LIN {X 0,Y 185.523,Z 180.554,A -85,B 0,C 180,E1 -22370.264,E2 -22370.264} C_VEL
LIN {X 0,Y 186.732,Z 185.626,A -85,B 0,C 180,E1 -22372.872,E2 -22372.872} C_VEL
LIN {X 0,Y 194.907,Z 207.144,A -85,B 0,C 180,E1 -22375.125,E2 -22375.125} C_VEL
LIN {X 0,Y 199.126,Z 220.308,A -85,B 0,C 180,E1 -22376.315,E2 -22376.315} C_VEL
LIN {X 0,Y 201.437,Z 240.888,A -85,B 0,C 180,E1 -22377.565,E2 -22377.565} C_VEL
LIN {X 0,Y 199.217,Z 285.056,A -85,B 0,C 180,E1 -22379.362,E2 -22379.362} C_VEL
LIN {X 0,Y 198.176,Z 290.854,A -85,B 0,C 180,E1 -22379.532,E2 -22379.532} C_VEL
LIN {X 0,Y 194.625,Z 300.116,A -85,B 0,C 180,E1 -22379.764,E2 -22379.764} C_VEL
LIN {X 0,Y 190.969,Z 309.221,A -85,B 0,C 180,E1 -22380.201,E2 -22380.201} C_VEL
LIN {X 0,Y 189.736,Z 314.767,A -85,B 0,C 180,E1 -22380.703,E2 -22380.703} C_VEL
LIN {X 0,Y 187.977,Z 326.317,A -85,B 0,C 180,E1 -22382.138,E2 -22382.138} C_VEL
LIN {X 0,Y 185.921,Z 337.434,A -85,B 0,C 180,E1 -22383.932,E2 -22383.932} C_VEL
LIN {X 0,Y 183.615,Z 348.891,A -85,B 0,C 180,E1 -22386.303,E2 -22386.303} C_VEL
LIN {X 0,Y 181.324,Z 359.447,A -85,B 0,C 180,E1 -22389.126,E2 -22389.126} C_VEL
LIN {X 0,Y 179.446,Z 368.889,A -85,B 0,C 180,E1 -22392.33,E2 -22392.33} C_VEL
LIN {X 0,Y 177.807,Z 376.667,A -85,B 0,C 180,E1 -22395.698,E2 -22395.698} C_VEL
LIN {X 0,Y 176.949,Z 381.981,A -85,B 0,C 180,E1 -22398.545,E2 -22398.545} C_VEL
LIN {X 0,Y 176.345,Z 387.087,A -85,B 0,C 180,E1 -22401.982,E2 -22401.982} C_VEL
LIN {X 0,Y 176.061,Z 390.987,A -85,B 0,C 180,E1 -22405.421,E2 -22405.421} C_VEL
LIN {X 0,Y 176.043,Z 392.971,A -85,B 0,C 180,E1 -22407.712,E2 -22407.712} C_VEL
LIN {X 0,Y 176.191,Z 394.524,A -85,B 0,C 180,E1 -22410,E2 -22410} C_VEL
LIN {X 0,Y 175.998,Z 395.943,A -85,B 0,C 180,E1 -22413.319,E2 -22413.319} C_VEL
LIN {X 0,Y 176.144,Z 396.529,A -85,B 0,C 180,E1 -22416.874,E2 -22416.874} C_VEL
LIN {X 0,Y 177.087,Z 395.919,A -85,B 0,C 180,E1 -22421.445,E2 -22421.445} C_VEL
LIN {X 0,Y 178.986,Z 393.704,A -85,B 0,C 180,E1 -22425.953,E2 -22425.953} C_VEL
LIN {X 0,Y 181.258,Z 391.001,A -85,B 0,C 180,E1 -22429.242,E2 -22429.242} C_VEL
LIN {X 0,Y 184.177,Z 387.313,A -85,B 0,C 180,E1 -22432.431,E2 -22432.431} C_VEL
LIN {X 0,Y 187.917,Z 381.869,A -85,B 0,C 180,E1 -22435.953,E2 -22435.953} C_VEL
LIN {X 0,Y 192.068,Z 375.591,A -85,B 0,C 180,E1 -22439.001,E2 -22439.001} C_VEL
LIN {X 0,Y 196.577,Z 368.083,A -85,B 0,C 180,E1 -22441.825,E2 -22441.825} C_VEL
LIN {X 0,Y 201.898,Z 358.701,A -85,B 0,C 180,E1 -22444.447,E2 -22444.447} C_VEL
LIN {X 0,Y 207.006,Z 348.132,A -85,B 0,C 180,E1 -22446.753,E2 -22446.753} C_VEL
LIN {X 0,Y 211.458,Z 337.471,A -85,B 0,C 180,E1 -22448.547,E2 -22448.547} C_VEL
LIN {X 0,Y 215.19,Z 327.2,A -85,B 0,C 180,E1 -22449.861,E2 -22449.861} C_VEL
LIN {X 0,Y 219.022,Z 314.154,A -85,B 0,C 180,E1 -22451.132,E2 -22451.132} C_VEL
LIN {X 0,Y 221.965,Z 300.978,A -85,B 0,C 180,E1 -22452.032,E2 -22452.032} C_VEL
LIN {X 0,Y 224.04,Z 287.051,A -85,B 0,C 180,E1 -22452.66,E2 -22452.66} C_VEL
LIN {X 0,Y 227.25,Z 253.842,A -85,B 0,C 180,E1 -22453.843,E2 -22453.843} C_VEL
LIN {X 0,Y 223.841,Z 244.653,A -85,B 0,C 180,E1 -22456.051,E2 -22456.051} C_VEL
LIN {X 0,Y 220.21,Z 236.597,A -85,B 0,C 180,E1 -22458.58,E2 -22458.58} C_VEL
LIN {X 0,Y 217.139,Z 230.6,A -85,B 0,C 180,E1 -22461.012,E2 -22461.012} C_VEL
LIN {X 0,Y 214.883,Z 226.367,A -85,B 0,C 180,E1 -22463.117,E2 -22463.117} C_VEL
LIN {X 0,Y 212.143,Z 221.304,A -85,B 0,C 180,E1 -22466.228,E2 -22466.228} C_VEL
LIN {X 0,Y 208.997,Z 215.881,A -85,B 0,C 180,E1 -22471.764,E2 -22471.764} C_VEL
LIN {X 0,Y 208.244,Z 214.671,A -85,B 0,C 180,E1 -22474.351,E2 -22474.351} C_VEL
LIN {X 0,Y 207.997,Z 214.147,A -85,B 0,C 180,E1 -22478.18,E2 -22478.18} C_VEL
LIN {X 0,Y 208.898,Z 214.551,A -85,B 0,C 180,E1 -22482.075,E2 -22482.075} C_VEL
LIN {X 0,Y 212.652,Z 219.409,A -85,B 0,C 180,E1 -22488.471,E2 -22488.471} C_VEL
LIN {X 0,Y 215.724,Z 224.28,A -85,B 0,C 180,E1 -22491.751,E2 -22491.751} C_VEL
LIN {X 0,Y 218.763,Z 228.903,A -85,B 0,C 180,E1 -22494.313,E2 -22494.313} C_VEL
LIN {X 0,Y 221.395,Z 233.953,A -85,B 0,C 180,E1 -22496.315,E2 -22496.315} C_VEL
LIN {X 0,Y 225.254,Z 241.753,A -85,B 0,C 180,E1 -22498.857,E2 -22498.857} C_VEL
LIN {X 0,Y 227.673,Z 247.671,A -85,B 0,C 180,E1 -22500.375,E2 -22500.375} C_VEL
LIN {X 0,Y 223.79,Z 286.154,A -85,B 0,C 180,E1 -22501.764,E2 -22501.764} C_VEL
LIN {X 0,Y 221.454,Z 299.905,A -85,B 0,C 180,E1 -22502.557,E2 -22502.557} C_VEL
LIN {X 0,Y 218.622,Z 311.882,A -85,B 0,C 180,E1 -22503.551,E2 -22503.551} C_VEL
LIN {X 0,Y 214.983,Z 323.909,A -85,B 0,C 180,E1 -22504.922,E2 -22504.922} C_VEL
LIN {X 0,Y 210.876,Z 334.991,A -85,B 0,C 180,E1 -22506.567,E2 -22506.567} C_VEL
LIN {X 0,Y 206.146,Z 345.721,A -85,B 0,C 180,E1 -22508.638,E2 -22508.638} C_VEL
LIN {X 0,Y 201.058,Z 355.6,A -85,B 0,C 180,E1 -22511.104,E2 -22511.104} C_VEL
LIN {X 0,Y 196.477,Z 363.559,A -85,B 0,C 180,E1 -22513.686,E2 -22513.686} C_VEL
LIN {X 0,Y 192.193,Z 370.197,A -85,B 0,C 180,E1 -22516.462,E2 -22516.462} C_VEL
LIN {X 0,Y 187.993,Z 376.022,A -85,B 0,C 180,E1 -22519.66,E2 -22519.66} C_VEL
LIN {X 0,Y 183.991,Z 381.142,A -85,B 0,C 180,E1 -22523.548,E2 -22523.548} C_VEL
LIN {X 0,Y 180.556,Z 384.879,A -85,B 0,C 180,E1 -22527.844,E2 -22527.844} C_VEL
LIN {X 0,Y 178.835,Z 386.437,A -85,B 0,C 180,E1 -22530.722,E2 -22530.722} C_VEL
LIN {X 0,Y 177.473,Z 387.301,A -85,B 0,C 180,E1 -22533.737,E2 -22533.737} C_VEL
LIN {X 0,Y 176.381,Z 387.452,A -85,B 0,C 180,E1 -22537.165,E2 -22537.165} C_VEL
LIN {X 0,Y 175.726,Z 386.737,A -85,B 0,C 180,E1 -22540.547,E2 -22540.547} C_VEL
LIN {X 0,Y 175.548,Z 385.172,A -85,B 0,C 180,E1 -22543.895,E2 -22543.895} C_VEL
LIN {X 0,Y 175.859,Z 381.648,A -85,B 0,C 180,E1 -22548.349,E2 -22548.349} C_VEL
LIN {X 0,Y 176.378,Z 377.958,A -85,B 0,C 180,E1 -22551.618,E2 -22551.618} C_VEL
LIN {X 0,Y 177.417,Z 371.966,A -85,B 0,C 180,E1 -22555.628,E2 -22555.628} C_VEL
LIN {X 0,Y 178.782,Z 364.796,A -85,B 0,C 180,E1 -22559.268,E2 -22559.268} C_VEL
LIN {X 0,Y 180.648,Z 355.985,A -85,B 0,C 180,E1 -22562.768,E2 -22562.768} C_VEL
LIN {X 0,Y 182.436,Z 347.714,A -85,B 0,C 180,E1 -22565.39,E2 -22565.39} C_VEL
LIN {X 0,Y 184.503,Z 337.858,A -85,B 0,C 180,E1 -22567.905,E2 -22567.905} C_VEL
LIN {X 0,Y 186.713,Z 326.401,A -85,B 0,C 180,E1 -22570.22,E2 -22570.22} C_VEL
LIN {X 0,Y 188.707,Z 314.366,A -85,B 0,C 180,E1 -22572.107,E2 -22572.107} C_VEL
LIN {X 0,Y 190.466,Z 301.472,A -85,B 0,C 180,E1 -22573.609,E2 -22573.609} C_VEL
LIN {X 0,Y 191.829,Z 288.229,A -85,B 0,C 180,E1 -22574.704,E2 -22574.704} C_VEL
LIN {X 0,Y 192.829,Z 272.096,A -85,B 0,C 180,E1 -22575.515,E2 -22575.515} C_VEL
LIN {X 0,Y 195.507,Z 223.333,A -85,B 0,C 180,E1 -22577.545,E2 -22577.545} C_VEL
LIN {X 0,Y 188.439,Z 202.79,A -85,B 0,C 180,E1 -22579.515,E2 -22579.515} C_VEL
LIN {X 0,Y 179.852,Z 183.966,A -85,B 0,C 180,E1 -22581.822,E2 -22581.822} C_VEL
LIN {X 0,Y 178.904,Z 181.199,A -85,B 0,C 180,E1 -22582.169,E2 -22582.169} C_VEL
LIN {X 0,Y 179.121,Z 181.175,A -85,B 0,C 180,E1 -22587.752,E2 -22587.752} C_VEL
LIN {X 0,Y 179.341,Z 181.15,A -85,B 0,C 180,E1 -22590,E2 -22590} C_VEL
LIN {X 0,Y 178.827,Z 181.214,A -85,B 0,C 180,E1 -22594.508,E2 -22594.508} C_VEL
LIN {X 0,Y 178.903,Z 181.203,A -85,B 0,C 180,E1 -22599.041,E2 -22599.041} C_VEL
LIN {X 0,Y 178.623,Z 181.236,A -85,B 0,C 180,E1 -22603.655,E2 -22603.655} C_VEL
LIN {X 0,Y 178.552,Z 181.244,A -85,B 0,C 180,E1 -22609.152,E2 -22609.152} C_VEL
LIN {X 0,Y 178.462,Z 181.253,A -85,B 0,C 180,E1 -22615.076,E2 -22615.076} C_VEL
LIN {X 0,Y 178.457,Z 181.247,A -85,B 0,C 180,E1 -22620.795,E2 -22620.795} C_VEL
LIN {X 0,Y 178.48,Z 181.247,A -85,B 0,C 180,E1 -22624.218,E2 -22624.218} C_VEL
LIN {X 0,Y 178.384,Z 181.263,A -85,B 0,C 180,E1 -22629.077,E2 -22629.077} C_VEL
LIN {X 0,Y 178.39,Z 181.25,A -85,B 0,C 180,E1 -22632.047,E2 -22632.047} C_VEL
LIN {X 0,Y 178.388,Z 181.253,A -85,B 0,C 180,E1 -22635.166,E2 -22635.166} C_VEL
LIN {X 0,Y 178.394,Z 181.261,A -85,B 0,C 180,E1 -22638.462,E2 -22638.462} C_VEL
LIN {X 0,Y 178.416,Z 181.251,A -85,B 0,C 180,E1 -22643.783,E2 -22643.783} C_VEL
LIN {X 0,Y 178.481,Z 181.231,A -85,B 0,C 180,E1 -22646.547,E2 -22646.547} C_VEL
LIN {X 0,Y 178.436,Z 181.255,A -85,B 0,C 180,E1 -22651.795,E2 -22651.795} C_VEL
LIN {X 0,Y 178.456,Z 181.251,A -85,B 0,C 180,E1 -22656.809,E2 -22656.809} C_VEL
LIN {X 0,Y 178.603,Z 181.212,A -85,B 0,C 180,E1 -22661.652,E2 -22661.652} C_VEL
LIN {X 0,Y 178.622,Z 181.23,A -85,B 0,C 180,E1 -22666.346,E2 -22666.346} C_VEL
LIN {X 0,Y 178.899,Z 181.193,A -85,B 0,C 180,E1 -22670.96,E2 -22670.96} C_VEL
LIN {X 0,Y 179.117,Z 181.163,A -85,B 0,C 180,E1 -22677.752,E2 -22677.752} C_VEL
LIN {X 0,Y 179.342,Z 181.143,A -85,B 0,C 180,E1 -22680.001,E2 -22680.001} C_VEL
LIN {X 0,Y 178.823,Z 181.202,A -85,B 0,C 180,E1 -22684.509,E2 -22684.509} C_VEL
LIN {X 0,Y 178.9,Z 181.193,A -85,B 0,C 180,E1 -22689.042,E2 -22689.042} C_VEL
LIN {X 0,Y 178.623,Z 181.234,A -85,B 0,C 180,E1 -22693.656,E2 -22693.656} C_VEL
LIN {X 0,Y 178.554,Z 181.241,A -85,B 0,C 180,E1 -22699.153,E2 -22699.153} C_VEL
LIN {X 0,Y 178.464,Z 181.249,A -85,B 0,C 180,E1 -22705.076,E2 -22705.076} C_VEL
LIN {X 0,Y 178.45,Z 181.252,A -85,B 0,C 180,E1 -22710.797,E2 -22710.797} C_VEL
LIN {X 0,Y 178.483,Z 181.236,A -85,B 0,C 180,E1 -22714.219,E2 -22714.219} C_VEL
LIN {X 0,Y 178.388,Z 181.264,A -85,B 0,C 180,E1 -22719.078,E2 -22719.078} C_VEL
LIN {X 0,Y 178.394,Z 181.264,A -85,B 0,C 180,E1 -22722.048,E2 -22722.048} C_VEL
LIN {X 0,Y 178.392,Z 181.264,A -85,B 0,C 180,E1 -22725.166,E2 -22725.166} C_VEL
LIN {X 0,Y 178.428,Z 181.35,A -85,B 0,C 180,E1 -22729.527,E2 -22729.527} C_VEL
LIN {X 0,Y 179.396,Z 185.381,A -85,B 0,C 180,E1 -22731.698,E2 -22731.698} C_VEL
LIN {X 0,Y 187.05,Z 205.093,A -85,B 0,C 180,E1 -22733.929,E2 -22733.929} C_VEL
LIN {X 0,Y 192.645,Z 221.29,A -85,B 0,C 180,E1 -22735.514,E2 -22735.514} C_VEL
LIN {X 0,Y 194.853,Z 241.898,A -85,B 0,C 180,E1 -22736.806,E2 -22736.806} C_VEL
LIN {X 0,Y 191.966,Z 293.825,A -85,B 0,C 180,E1 -22739.019,E2 -22739.019} C_VEL
LIN {X 0,Y 190.668,Z 307.543,A -85,B 0,C 180,E1 -22740.006,E2 -22740.006} C_VEL
LIN {X 0,Y 189.736,Z 314.767,A -85,B 0,C 180,E1 -22740.703,E2 -22740.703} C_VEL
LIN {X 0,Y 188.42,Z 320.204,A -85,B 0,C 180,E1 -22741.268,E2 -22741.268} C_VEL
LIN {X 0,Y 184.29,Z 328.708,A -85,B 0,C 180,E1 -22742.179,E2 -22742.179} C_VEL
LIN {X 0,Y 179.879,Z 336.864,A -85,B 0,C 180,E1 -22743.32,E2 -22743.32} C_VEL
LIN {X 0,Y 178.153,Z 341.765,A -85,B 0,C 180,E1 -22744.235,E2 -22744.235} C_VEL
LIN {X 0,Y 175.795,Z 352.848,A -85,B 0,C 180,E1 -22746.856,E2 -22746.856} C_VEL
LIN {X 0,Y 174.039,Z 361.107,A -85,B 0,C 180,E1 -22749.308,E2 -22749.308} C_VEL
LIN {X 0,Y 172.038,Z 370.429,A -85,B 0,C 180,E1 -22752.772,E2 -22752.772} C_VEL
LIN {X 0,Y 170.499,Z 377.896,A -85,B 0,C 180,E1 -22756.289,E2 -22756.289} C_VEL
LIN {X 0,Y 169.695,Z 382.937,A -85,B 0,C 180,E1 -22759.259,E2 -22759.259} C_VEL
LIN {X 0,Y 169.191,Z 387.794,A -85,B 0,C 180,E1 -22762.841,E2 -22762.841} C_VEL
LIN {X 0,Y 168.933,Z 391.821,A -85,B 0,C 180,E1 -22766.834,E2 -22766.834} C_VEL
LIN {X 0,Y 169.114,Z 394.051,A -85,B 0,C 180,E1 -22770,E2 -22770} C_VEL
LIN {X 0,Y 168.932,Z 395.495,A -85,B 0,C 180,E1 -22773.163,E2 -22773.163} C_VEL
LIN {X 0,Y 169.097,Z 396.296,A -85,B 0,C 180,E1 -22777.162,E2 -22777.162} C_VEL
LIN {X 0,Y 170.111,Z 395.823,A -85,B 0,C 180,E1 -22781.921,E2 -22781.921} C_VEL
LIN {X 0,Y 171.013,Z 395.023,A -85,B 0,C 180,E1 -22784.274,E2 -22784.274} C_VEL
LIN {X 0,Y 172.144,Z 393.803,A -85,B 0,C 180,E1 -22786.605,E2 -22786.605} C_VEL
LIN {X 0,Y 175.512,Z 390.163,A -85,B 0,C 180,E1 -22791.123,E2 -22791.123} C_VEL
LIN {X 0,Y 178.852,Z 386.299,A -85,B 0,C 180,E1 -22794.367,E2 -22794.367} C_VEL
LIN {X 0,Y 182.323,Z 381.399,A -85,B 0,C 180,E1 -22797.552,E2 -22797.552} C_VEL
LIN {X 0,Y 186.734,Z 375.257,A -85,B 0,C 180,E1 -22800.536,E2 -22800.536} C_VEL
LIN {X 0,Y 191.548,Z 367.741,A -85,B 0,C 180,E1 -22803.391,E2 -22803.391} C_VEL
LIN {X 0,Y 197.127,Z 358.396,A -85,B 0,C 180,E1 -22806.033,E2 -22806.033} C_VEL
LIN {X 0,Y 202.496,Z 347.857,A -85,B 0,C 180,E1 -22808.343,E2 -22808.343} C_VEL
LIN {X 0,Y 207.165,Z 337.161,A -85,B 0,C 180,E1 -22810.132,E2 -22810.132} C_VEL
LIN {X 0,Y 211.624,Z 325.18,A -85,B 0,C 180,E1 -22811.62,E2 -22811.62} C_VEL
LIN {X 0,Y 215.359,Z 312.674,A -85,B 0,C 180,E1 -22812.779,E2 -22812.779} C_VEL
LIN {X 0,Y 218.437,Z 298.841,A -85,B 0,C 180,E1 -22813.679,E2 -22813.679} C_VEL
LIN {X 0,Y 220.466,Z 284.829,A -85,B 0,C 180,E1 -22814.28,E2 -22814.28} C_VEL
LIN {X 0,Y 223.268,Z 256.597,A -85,B 0,C 180,E1 -22815.324,E2 -22815.324} C_VEL
LIN {X 0,Y 220.341,Z 248.569,A -85,B 0,C 180,E1 -22817.388,E2 -22817.388} C_VEL
LIN {X 0,Y 216.972,Z 240.885,A -85,B 0,C 180,E1 -22820.019,E2 -22820.019} C_VEL
LIN {X 0,Y 214.617,Z 236.021,A -85,B 0,C 180,E1 -22822.098,E2 -22822.098} C_VEL
LIN {X 0,Y 212.784,Z 232.436,A -85,B 0,C 180,E1 -22823.967,E2 -22823.967} C_VEL
LIN {X 0,Y 210.54,Z 227.94,A -85,B 0,C 180,E1 -22826.763,E2 -22826.763} C_VEL
LIN {X 0,Y 207.662,Z 222.626,A -85,B 0,C 180,E1 -22832.277,E2 -22832.277} C_VEL
LIN {X 0,Y 207.005,Z 221.519,A -85,B 0,C 180,E1 -22835.002,E2 -22835.002} C_VEL
LIN {X 0,Y 207.196,Z 221.214,A -85,B 0,C 180,E1 -22840.171,E2 -22840.171} C_VEL
LIN {X 0,Y 207.826,Z 221.735,A -85,B 0,C 180,E1 -22842.28,E2 -22842.28} C_VEL
LIN {X 0,Y 211.159,Z 226.339,A -85,B 0,C 180,E1 -22848.115,E2 -22848.115} C_VEL
LIN {X 0,Y 213.886,Z 230.84,A -85,B 0,C 180,E1 -22851.197,E2 -22851.197} C_VEL
LIN {X 0,Y 216.591,Z 235.183,A -85,B 0,C 180,E1 -22853.648,E2 -22853.648} C_VEL
LIN {X 0,Y 219.433,Z 241.032,A -85,B 0,C 180,E1 -22855.921,E2 -22855.921} C_VEL
LIN {X 0,Y 222.35,Z 247.28,A -85,B 0,C 180,E1 -22857.978,E2 -22857.978} C_VEL
LIN {X 0,Y 223.761,Z 251.117,A -85,B 0,C 180,E1 -22858.95,E2 -22858.95} C_VEL
LIN {X 0,Y 219.931,Z 286.55,A -85,B 0,C 180,E1 -22860.23,E2 -22860.23} C_VEL
LIN {X 0,Y 217.492,Z 300.162,A -85,B 0,C 180,E1 -22861.017,E2 -22861.017} C_VEL
LIN {X 0,Y 214.313,Z 312.803,A -85,B 0,C 180,E1 -22862.079,E2 -22862.079} C_VEL
LIN {X 0,Y 210.618,Z 324.429,A -85,B 0,C 180,E1 -22863.414,E2 -22863.414} C_VEL
LIN {X 0,Y 206.079,Z 336.077,A -85,B 0,C 180,E1 -22865.159,E2 -22865.159} C_VEL
LIN {X 0,Y 201.067,Z 346.77,A -85,B 0,C 180,E1 -22867.278,E2 -22867.278} C_VEL
LIN {X 0,Y 195.624,Z 356.675,A -85,B 0,C 180,E1 -22869.824,E2 -22869.824} C_VEL
LIN {X 0,Y 191.053,Z 364.048,A -85,B 0,C 180,E1 -22872.304,E2 -22872.304} C_VEL
LIN {X 0,Y 186.224,Z 371,A -85,B 0,C 180,E1 -22875.317,E2 -22875.317} C_VEL
LIN {X 0,Y 181.178,Z 377.479,A -85,B 0,C 180,E1 -22879.104,E2 -22879.104} C_VEL
LIN {X 0,Y 178.066,Z 381.099,A -85,B 0,C 180,E1 -22882.02,E2 -22882.02} C_VEL
LIN {X 0,Y 174.376,Z 384.854,A -85,B 0,C 180,E1 -22886.316,E2 -22886.316} C_VEL
LIN {X 0,Y 171.67,Z 386.998,A -85,B 0,C 180,E1 -22890.717,E2 -22890.717} C_VEL
LIN {X 0,Y 169.726,Z 387.734,A -85,B 0,C 180,E1 -22895.429,E2 -22895.429} C_VEL
LIN {X 0,Y 168.922,Z 387.306,A -85,B 0,C 180,E1 -22898.613,E2 -22898.613} C_VEL
LIN {X 0,Y 168.516,Z 386.174,A -85,B 0,C 180,E1 -22901.856,E2 -22901.856} C_VEL
LIN {X 0,Y 168.447,Z 384.252,A -85,B 0,C 180,E1 -22905.175,E2 -22905.175} C_VEL
LIN {X 0,Y 168.787,Z 381.419,A -85,B 0,C 180,E1 -22908.545,E2 -22908.545} C_VEL
LIN {X 0,Y 169.35,Z 377.474,A -85,B 0,C 180,E1 -22912.043,E2 -22912.043} C_VEL
LIN {X 0,Y 170.284,Z 372.225,A -85,B 0,C 180,E1 -22915.631,E2 -22915.631} C_VEL
LIN {X 0,Y 171.64,Z 365.335,A -85,B 0,C 180,E1 -22919.3,E2 -22919.3} C_VEL
LIN {X 0,Y 173.547,Z 356.471,A -85,B 0,C 180,E1 -22922.986,E2 -22922.986} C_VEL
LIN {X 0,Y 175.713,Z 346.879,A -85,B 0,C 180,E1 -22926.112,E2 -22926.112} C_VEL
LIN {X 0,Y 178.027,Z 336.047,A -85,B 0,C 180,E1 -22928.886,E2 -22928.886} C_VEL
LIN {X 0,Y 180.053,Z 325.747,A -85,B 0,C 180,E1 -22930.979,E2 -22930.979} C_VEL
LIN {X 0,Y 182.068,Z 313.748,A -85,B 0,C 180,E1 -22932.881,E2 -22932.881} C_VEL
LIN {X 0,Y 183.766,Z 301.825,A -85,B 0,C 180,E1 -22934.303,E2 -22934.303} C_VEL
LIN {X 0,Y 185.124,Z 288.738,A -85,B 0,C 180,E1 -22935.434,E2 -22935.434} C_VEL
LIN {X 0,Y 186.186,Z 273.821,A -85,B 0,C 180,E1 -22936.216,E2 -22936.216} C_VEL
LIN {X 0,Y 188.893,Z 224.499,A -85,B 0,C 180,E1 -22938.349,E2 -22938.349} C_VEL
LIN {X 0,Y 182.114,Z 204.991,A -85,B 0,C 180,E1 -22940.338,E2 -22940.338} C_VEL
LIN {X 0,Y 174.085,Z 187.342,A -85,B 0,C 180,E1 -22942.607,E2 -22942.607} C_VEL
LIN {X 0,Y 171.926,Z 182.6,A -85,B 0,C 180,E1 -22943.251,E2 -22943.251} C_VEL
LIN {X 0,Y 171.837,Z 182.08,A -85,B 0,C 180,E1 -22943.395,E2 -22943.395} C_VEL
LIN {X 0,Y 172.306,Z 182.026,A -85,B 0,C 180,E1 -22950,E2 -22950} C_VEL
LIN {X 0,Y 171.777,Z 182.092,A -85,B 0,C 180,E1 -22954.694,E2 -22954.694} C_VEL
LIN {X 0,Y 171.841,Z 182.084,A -85,B 0,C 180,E1 -22959.416,E2 -22959.416} C_VEL
LIN {X 0,Y 171.539,Z 182.119,A -85,B 0,C 180,E1 -22964.231,E2 -22964.231} C_VEL
LIN {X 0,Y 171.475,Z 182.126,A -85,B 0,C 180,E1 -22969.499,E2 -22969.499} C_VEL
LIN {X 0,Y 171.4,Z 182.134,A -85,B 0,C 180,E1 -22975.57,E2 -22975.57} C_VEL
LIN {X 0,Y 171.414,Z 182.125,A -85,B 0,C 180,E1 -22980.573,E2 -22980.573} C_VEL
LIN {X 0,Y 171.389,Z 182.132,A -85,B 0,C 180,E1 -22985.035,E2 -22985.035} C_VEL
LIN {X 0,Y 171.34,Z 182.141,A -85,B 0,C 180,E1 -22988.801,E2 -22988.801} C_VEL
LIN {X 0,Y 171.315,Z 182.129,A -85,B 0,C 180,E1 -22994.219,E2 -22994.219} C_VEL
LIN {X 0,Y 171.326,Z 182.144,A -85,B 0,C 180,E1 -22998.98,E2 -22998.98} C_VEL
LIN {X 0,Y 171.357,Z 182.136,A -85,B 0,C 180,E1 -23002.034,E2 -23002.034} C_VEL
LIN {X 0,Y 171.395,Z 182.118,A -85,B 0,C 180,E1 -23005.094,E2 -23005.094} C_VEL
LIN {X 0,Y 171.405,Z 182.127,A -85,B 0,C 180,E1 -23010.527,E2 -23010.527} C_VEL
LIN {X 0,Y 171.399,Z 182.132,A -85,B 0,C 180,E1 -23015.794,E2 -23015.794} C_VEL
LIN {X 0,Y 171.505,Z 182.096,A -85,B 0,C 180,E1 -23020.864,E2 -23020.864} C_VEL
LIN {X 0,Y 171.538,Z 182.11,A -85,B 0,C 180,E1 -23025.771,E2 -23025.771} C_VEL
LIN {X 0,Y 171.838,Z 182.074,A -85,B 0,C 180,E1 -23030.585,E2 -23030.585} C_VEL
LIN {X 0,Y 171.771,Z 182.066,A -85,B 0,C 180,E1 -23035.307,E2 -23035.307} C_VEL
LIN {X 0,Y 172.306,Z 182.019,A -85,B 0,C 180,E1 -23040.001,E2 -23040.001} C_VEL
LIN {X 0,Y 171.773,Z 182.079,A -85,B 0,C 180,E1 -23044.695,E2 -23044.695} C_VEL
LIN {X 0,Y 171.839,Z 182.073,A -85,B 0,C 180,E1 -23049.417,E2 -23049.417} C_VEL
LIN {X 0,Y 171.538,Z 182.114,A -85,B 0,C 180,E1 -23054.231,E2 -23054.231} C_VEL
LIN {X 0,Y 171.478,Z 182.124,A -85,B 0,C 180,E1 -23059.499,E2 -23059.499} C_VEL
LIN {X 0,Y 171.401,Z 182.131,A -85,B 0,C 180,E1 -23065.569,E2 -23065.569} C_VEL
LIN {X 0,Y 171.406,Z 182.131,A -85,B 0,C 180,E1 -23070.567,E2 -23070.567} C_VEL
LIN {X 0,Y 171.393,Z 182.123,A -85,B 0,C 180,E1 -23075.036,E2 -23075.036} C_VEL
LIN {X 0,Y 171.344,Z 182.142,A -85,B 0,C 180,E1 -23078.802,E2 -23078.802} C_VEL
LIN {X 0,Y 171.319,Z 182.146,A -85,B 0,C 180,E1 -23084.219,E2 -23084.219} C_VEL
LIN {X 0,Y 171.389,Z 182.155,A -85,B 0,C 180,E1 -23088.772,E2 -23088.772} C_VEL
LIN {X 0,Y 172.07,Z 185.224,A -85,B 0,C 180,E1 -23090.448,E2 -23090.448} C_VEL
LIN {X 0,Y 179.137,Z 202.761,A -85,B 0,C 180,E1 -23092.605,E2 -23092.605} C_VEL
LIN {X 0,Y 185.907,Z 222.273,A -85,B 0,C 180,E1 -23094.653,E2 -23094.653} C_VEL
LIN {X 0,Y 187.097,Z 229.819,A -85,B 0,C 180,E1 -23095.205,E2 -23095.205} C_VEL
LIN {X 0,Y 188.269,Z 242.646,A -85,B 0,C 180,E1 -23096.01,E2 -23096.01} C_VEL
LIN {X 0,Y 185.356,Z 293.514,A -85,B 0,C 180,E1 -23098.259,E2 -23098.259} C_VEL
LIN {X 0,Y 184.001,Z 307.3,A -85,B 0,C 180,E1 -23099.279,E2 -23099.279} C_VEL
LIN {X 0,Y 182.368,Z 319.378,A -85,B 0,C 180,E1 -23100.571,E2 -23100.571} C_VEL
LIN {X 0,Y 180.071,Z 331.931,A -85,B 0,C 180,E1 -23102.389,E2 -23102.389} C_VEL
LIN {X 0,Y 178.153,Z 341.765,A -85,B 0,C 180,E1 -23104.235,E2 -23104.235} C_VEL
LIN {X 0,Y 176.447,Z 346.538,A -85,B 0,C 180,E1 -23105.227,E2 -23105.227} C_VEL
LIN {X 0,Y 172.025,Z 353.866,A -85,B 0,C 180,E1 -23106.88,E2 -23106.88} C_VEL
LIN {X 0,Y 167.702,Z 360.692,A -85,B 0,C 180,E1 -23108.817,E2 -23108.817} C_VEL
LIN {X 0,Y 166.185,Z 364.652,A -85,B 0,C 180,E1 -23110.227,E2 -23110.227} C_VEL
LIN {X 0,Y 164.605,Z 371.946,A -85,B 0,C 180,E1 -23113.25,E2 -23113.25} C_VEL
LIN {X 0,Y 163.209,Z 379.043,A -85,B 0,C 180,E1 -23116.934,E2 -23116.934} C_VEL
LIN {X 0,Y 162.287,Z 385.506,A -85,B 0,C 180,E1 -23121.282,E2 -23121.282} C_VEL
LIN {X 0,Y 161.932,Z 389.689,A -85,B 0,C 180,E1 -23125.02,E2 -23125.02} C_VEL
LIN {X 0,Y 161.888,Z 391.867,A -85,B 0,C 180,E1 -23127.511,E2 -23127.511} C_VEL
LIN {X 0,Y 162.038,Z 393.549,A -85,B 0,C 180,E1 -23130,E2 -23130} C_VEL
LIN {X 0,Y 161.853,Z 394.955,A -85,B 0,C 180,E1 -23132.894,E2 -23132.894} C_VEL
LIN {X 0,Y 162.029,Z 396.059,A -85,B 0,C 180,E1 -23137.476,E2 -23137.476} C_VEL
LIN {X 0,Y 163.157,Z 395.723,A -85,B 0,C 180,E1 -23142.437,E2 -23142.437} C_VEL
LIN {X 0,Y 165.329,Z 393.897,A -85,B 0,C 180,E1 -23147.311,E2 -23147.311} C_VEL
LIN {X 0,Y 166.987,Z 392.384,A -85,B 0,C 180,E1 -23149.675,E2 -23149.675} C_VEL
LIN {X 0,Y 170.015,Z 389.345,A -85,B 0,C 180,E1 -23153.122,E2 -23153.122} C_VEL
LIN {X 0,Y 173.561,Z 385.303,A -85,B 0,C 180,E1 -23156.45,E2 -23156.45} C_VEL
LIN {X 0,Y 177.571,Z 380.206,A -85,B 0,C 180,E1 -23159.651,E2 -23159.651} C_VEL
LIN {X 0,Y 182.405,Z 373.865,A -85,B 0,C 180,E1 -23162.643,E2 -23162.643} C_VEL
LIN {X 0,Y 186.684,Z 367.498,A -85,B 0,C 180,E1 -23165.036,E2 -23165.036} C_VEL
LIN {X 0,Y 192.518,Z 358.143,A -85,B 0,C 180,E1 -23167.695,E2 -23167.695} C_VEL
LIN {X 0,Y 198.144,Z 347.584,A -85,B 0,C 180,E1 -23170.006,E2 -23170.006} C_VEL
LIN {X 0,Y 203.021,Z 336.957,A -85,B 0,C 180,E1 -23171.787,E2 -23171.787} C_VEL
LIN {X 0,Y 207.685,Z 325.055,A -85,B 0,C 180,E1 -23173.254,E2 -23173.254} C_VEL
LIN {X 0,Y 211.273,Z 313.725,A -85,B 0,C 180,E1 -23174.311,E2 -23174.311} C_VEL
LIN {X 0,Y 214.47,Z 300.41,A -85,B 0,C 180,E1 -23175.212,E2 -23175.212} C_VEL
LIN {X 0,Y 216.736,Z 286.356,A -85,B 0,C 180,E1 -23175.83,E2 -23175.83} C_VEL
LIN {X 0,Y 219.482,Z 259.569,A -85,B 0,C 180,E1 -23176.84,E2 -23176.84} C_VEL
LIN {X 0,Y 217.301,Z 253.29,A -85,B 0,C 180,E1 -23178.567,E2 -23178.567} C_VEL
LIN {X 0,Y 214.252,Z 246.021,A -85,B 0,C 180,E1 -23181.161,E2 -23181.161} C_VEL
LIN {X 0,Y 212.348,Z 241.789,A -85,B 0,C 180,E1 -23183.065,E2 -23183.065} C_VEL
LIN {X 0,Y 210.913,Z 238.821,A -85,B 0,C 180,E1 -23184.633,E2 -23184.633} C_VEL
LIN {X 0,Y 208.866,Z 234.483,A -85,B 0,C 180,E1 -23187.426,E2 -23187.426} C_VEL
LIN {X 0,Y 206.346,Z 229.374,A -85,B 0,C 180,E1 -23192.788,E2 -23192.788} C_VEL
LIN {X 0,Y 205.772,Z 228.371,A -85,B 0,C 180,E1 -23195.804,E2 -23195.804} C_VEL
LIN {X 0,Y 206.31,Z 228.334,A -85,B 0,C 180,E1 -23201.172,E2 -23201.172} C_VEL
LIN {X 0,Y 207.122,Z 229.711,A -85,B 0,C 180,E1 -23203.465,E2 -23203.465} C_VEL
LIN {X 0,Y 209.625,Z 233.092,A -85,B 0,C 180,E1 -23207.67,E2 -23207.67} C_VEL
LIN {X 0,Y 211.969,Z 237.247,A -85,B 0,C 180,E1 -23210.534,E2 -23210.534} C_VEL
LIN {X 0,Y 214.38,Z 241.282,A -85,B 0,C 180,E1 -23212.875,E2 -23212.875} C_VEL
LIN {X 0,Y 216.998,Z 247.043,A -85,B 0,C 180,E1 -23215.137,E2 -23215.137} C_VEL
LIN {X 0,Y 219.461,Z 252.674,A -85,B 0,C 180,E1 -23217.05,E2 -23217.05} C_VEL
LIN {X 0,Y 220.015,Z 254.15,A -85,B 0,C 180,E1 -23217.453,E2 -23217.453} C_VEL
LIN {X 0,Y 216.234,Z 287.473,A -85,B 0,C 180,E1 -23218.661,E2 -23218.661} C_VEL
LIN {X 0,Y 213.812,Z 300.27,A -85,B 0,C 180,E1 -23219.387,E2 -23219.387} C_VEL
LIN {X 0,Y 210.833,Z 311.927,A -85,B 0,C 180,E1 -23220.347,E2 -23220.347} C_VEL
LIN {X 0,Y 206.839,Z 324.068,A -85,B 0,C 180,E1 -23221.714,E2 -23221.714} C_VEL
LIN {X 0,Y 202.098,Z 335.694,A -85,B 0,C 180,E1 -23223.436,E2 -23223.436} C_VEL
LIN {X 0,Y 196.691,Z 346.702,A -85,B 0,C 180,E1 -23225.59,E2 -23225.59} C_VEL
LIN {X 0,Y 191.11,Z 356.456,A -85,B 0,C 180,E1 -23228.087,E2 -23228.087} C_VEL
LIN {X 0,Y 185.661,Z 364.773,A -85,B 0,C 180,E1 -23230.909,E2 -23230.909} C_VEL
LIN {X 0,Y 180.257,Z 371.983,A -85,B 0,C 180,E1 -23234.168,E2 -23234.168} C_VEL
LIN {X 0,Y 175.248,Z 377.911,A -85,B 0,C 180,E1 -23237.799,E2 -23237.799} C_VEL
LIN {X 0,Y 171.012,Z 382.398,A -85,B 0,C 180,E1 -23241.706,E2 -23241.706} C_VEL
LIN {X 0,Y 168.399,Z 384.806,A -85,B 0,C 180,E1 -23244.666,E2 -23244.666} C_VEL
LIN {X 0,Y 166.203,Z 386.5,A -85,B 0,C 180,E1 -23247.718,E2 -23247.718} C_VEL
LIN {X 0,Y 164.262,Z 387.621,A -85,B 0,C 180,E1 -23251.164,E2 -23251.164} C_VEL
LIN {X 0,Y 162.762,Z 387.939,A -85,B 0,C 180,E1 -23254.876,E2 -23254.876} C_VEL
LIN {X 0,Y 161.831,Z 387.357,A -85,B 0,C 180,E1 -23258.585,E2 -23258.585} C_VEL
LIN {X 0,Y 161.393,Z 385.904,A -85,B 0,C 180,E1 -23262.246,E2 -23262.246} C_VEL
LIN {X 0,Y 161.376,Z 383.631,A -85,B 0,C 180,E1 -23265.83,E2 -23265.83} C_VEL
LIN {X 0,Y 161.93,Z 379.421,A -85,B 0,C 180,E1 -23270.405,E2 -23270.405} C_VEL
LIN {X 0,Y 162.7,Z 374.955,A -85,B 0,C 180,E1 -23273.957,E2 -23273.957} C_VEL
LIN {X 0,Y 163.753,Z 369.334,A -85,B 0,C 180,E1 -23277.488,E2 -23277.488} C_VEL
LIN {X 0,Y 165.079,Z 363.009,A -85,B 0,C 180,E1 -23280.687,E2 -23280.687} C_VEL
LIN {X 0,Y 167.006,Z 354.548,A -85,B 0,C 180,E1 -23284.113,E2 -23284.113} C_VEL
LIN {X 0,Y 169.338,Z 344.57,A -85,B 0,C 180,E1 -23287.315,E2 -23287.315} C_VEL
LIN {X 0,Y 171.496,Z 334.758,A -85,B 0,C 180,E1 -23289.813,E2 -23289.813} C_VEL
LIN {X 0,Y 173.641,Z 323.774,A -85,B 0,C 180,E1 -23292.025,E2 -23292.025} C_VEL
LIN {X 0,Y 175.778,Z 311.181,A -85,B 0,C 180,E1 -23293.983,E2 -23293.983} C_VEL
LIN {X 0,Y 177.56,Z 298.182,A -85,B 0,C 180,E1 -23295.458,E2 -23295.458} C_VEL
LIN {X 0,Y 178.89,Z 283.878,A -85,B 0,C 180,E1 -23296.57,E2 -23296.57} C_VEL
LIN {X 0,Y 181.111,Z 248.12,A -85,B 0,C 180,E1 -23298.201,E2 -23298.201} C_VEL
LIN {X 0,Y 182.317,Z 225.866,A -85,B 0,C 180,E1 -23299.203,E2 -23299.203} C_VEL
LIN {X 0,Y 176.159,Z 208.076,A -85,B 0,C 180,E1 -23301.107,E2 -23301.107} C_VEL
LIN {X 0,Y 168.534,Z 191.154,A -85,B 0,C 180,E1 -23303.355,E2 -23303.355} C_VEL
LIN {X 0,Y 164.905,Z 183.853,A -85,B 0,C 180,E1 -23304.459,E2 -23304.459} C_VEL
LIN {X 0,Y 164.757,Z 182.963,A -85,B 0,C 180,E1 -23304.646,E2 -23304.646} C_VEL
LIN {X 0,Y 165.27,Z 182.903,A -85,B 0,C 180,E1 -23310,E2 -23310} C_VEL
LIN {X 0,Y 164.817,Z 182.957,A -85,B 0,C 180,E1 -23317.35,E2 -23317.35} C_VEL
LIN {X 0,Y 164.699,Z 182.972,A -85,B 0,C 180,E1 -23321.058,E2 -23321.058} C_VEL
LIN {X 0,Y 164.425,Z 183.003,A -85,B 0,C 180,E1 -23327.41,E2 -23327.41} C_VEL
LIN {X 0,Y 164.416,Z 183.003,A -85,B 0,C 180,E1 -23329.997,E2 -23329.997} C_VEL
LIN {X 0,Y 164.336,Z 183.014,A -85,B 0,C 180,E1 -23336.094,E2 -23336.094} C_VEL
LIN {X 0,Y 164.35,Z 183,A -85,B 0,C 180,E1 -23341.215,E2 -23341.215} C_VEL
LIN {X 0,Y 164.277,Z 183.021,A -85,B 0,C 180,E1 -23346.794,E2 -23346.794} C_VEL
LIN {X 0,Y 164.283,Z 183.015,A -85,B 0,C 180,E1 -23349.918,E2 -23349.918} C_VEL
LIN {X 0,Y 164.277,Z 183.003,A -85,B 0,C 180,E1 -23353.342,E2 -23353.342} C_VEL
LIN {X 0,Y 164.257,Z 183.018,A -85,B 0,C 180,E1 -23356.798,E2 -23356.798} C_VEL
LIN {X 0,Y 164.286,Z 183.02,A -85,B 0,C 180,E1 -23360.356,E2 -23360.356} C_VEL
LIN {X 0,Y 164.323,Z 183.003,A -85,B 0,C 180,E1 -23364.352,E2 -23364.352} C_VEL
LIN {X 0,Y 164.364,Z 182.997,A -85,B 0,C 180,E1 -23369.13,E2 -23369.13} C_VEL
LIN {X 0,Y 164.354,Z 183.012,A -85,B 0,C 180,E1 -23374.685,E2 -23374.685} C_VEL
LIN {X 0,Y 164.414,Z 182.983,A -85,B 0,C 180,E1 -23380.119,E2 -23380.119} C_VEL
LIN {X 0,Y 164.468,Z 182.99,A -85,B 0,C 180,E1 -23385.145,E2 -23385.145} C_VEL
LIN {X 0,Y 164.76,Z 182.958,A -85,B 0,C 180,E1 -23390.177,E2 -23390.177} C_VEL
LIN {X 0,Y 164.813,Z 182.941,A -85,B 0,C 180,E1 -23392.651,E2 -23392.651} C_VEL
LIN {X 0,Y 165.271,Z 182.895,A -85,B 0,C 180,E1 -23400.001,E2 -23400.001} C_VEL
LIN {X 0,Y 164.813,Z 182.938,A -85,B 0,C 180,E1 -23407.351,E2 -23407.351} C_VEL
LIN {X 0,Y 164.7,Z 182.967,A -85,B 0,C 180,E1 -23411.057,E2 -23411.057} C_VEL
LIN {X 0,Y 164.423,Z 182.993,A -85,B 0,C 180,E1 -23417.411,E2 -23417.411} C_VEL
LIN {X 0,Y 164.419,Z 183.006,A -85,B 0,C 180,E1 -23419.997,E2 -23419.997} C_VEL
LIN {X 0,Y 164.336,Z 183.016,A -85,B 0,C 180,E1 -23426.093,E2 -23426.093} C_VEL
LIN {X 0,Y 164.344,Z 183.004,A -85,B 0,C 180,E1 -23431.21,E2 -23431.21} C_VEL
LIN {X 0,Y 164.28,Z 183.019,A -85,B 0,C 180,E1 -23436.794,E2 -23436.794} C_VEL
LIN {X 0,Y 164.286,Z 183.018,A -85,B 0,C 180,E1 -23439.919,E2 -23439.919} C_VEL
LIN {X 0,Y 164.281,Z 183.022,A -85,B 0,C 180,E1 -23443.343,E2 -23443.343} C_VEL
LIN {X 0,Y 164.308,Z 183.027,A -85,B 0,C 180,E1 -23447.993,E2 -23447.993} C_VEL
LIN {X 0,Y 164.767,Z 185.015,A -85,B 0,C 180,E1 -23449.094,E2 -23449.094} C_VEL
LIN {X 0,Y 172.369,Z 203.596,A -85,B 0,C 180,E1 -23451.55,E2 -23451.55} C_VEL
LIN {X 0,Y 179.426,Z 223.731,A -85,B 0,C 180,E1 -23453.786,E2 -23453.786} C_VEL
LIN {X 0,Y 180.247,Z 228.001,A -85,B 0,C 180,E1 -23454.138,E2 -23454.138} C_VEL
LIN {X 0,Y 181.797,Z 242.264,A -85,B 0,C 180,E1 -23455.116,E2 -23455.116} C_VEL
LIN {X 0,Y 178.767,Z 293.265,A -85,B 0,C 180,E1 -23457.445,E2 -23457.445} C_VEL
LIN {X 0,Y 177.352,Z 307.043,A -85,B 0,C 180,E1 -23458.494,E2 -23458.494} C_VEL
LIN {X 0,Y 175.499,Z 320.162,A -85,B 0,C 180,E1 -23459.962,E2 -23459.962} C_VEL
LIN {X 0,Y 173.142,Z 332.485,A -85,B 0,C 180,E1 -23461.844,E2 -23461.844} C_VEL
LIN {X 0,Y 170.849,Z 343.677,A -85,B 0,C 180,E1 -23464.083,E2 -23464.083} C_VEL
LIN {X 0,Y 168.494,Z 354.193,A -85,B 0,C 180,E1 -23466.787,E2 -23466.787} C_VEL
LIN {X 0,Y 166.559,Z 362.99,A -85,B 0,C 180,E1 -23469.628,E2 -23469.628} C_VEL
LIN {X 0,Y 166.185,Z 364.652,A -85,B 0,C 180,E1 -23470.227,E2 -23470.227} C_VEL
LIN {X 0,Y 164.717,Z 368.493,A -85,B 0,C 180,E1 -23471.719,E2 -23471.719} C_VEL
LIN {X 0,Y 160.651,Z 374.032,A -85,B 0,C 180,E1 -23474.219,E2 -23474.219} C_VEL
LIN {X 0,Y 156.758,Z 379.046,A -85,B 0,C 180,E1 -23476.986,E2 -23476.986} C_VEL
LIN {X 0,Y 155.601,Z 381.869,A -85,B 0,C 180,E1 -23478.852,E2 -23478.852} C_VEL
LIN {X 0,Y 154.973,Z 387.667,A -85,B 0,C 180,E1 -23483.49,E2 -23483.49} C_VEL
LIN {X 0,Y 154.818,Z 391.24,A -85,B 0,C 180,E1 -23487.398,E2 -23487.398} C_VEL
LIN {X 0,Y 154.945,Z 393.044,A -85,B 0,C 180,E1 -23490,E2 -23490} C_VEL
LIN {X 0,Y 154.795,Z 394.402,A -85,B 0,C 180,E1 -23492.733,E2 -23492.733} C_VEL
LIN {X 0,Y 154.975,Z 395.768,A -85,B 0,C 180,E1 -23497.819,E2 -23497.819} C_VEL
LIN {X 0,Y 155.45,Z 395.905,A -85,B 0,C 180,E1 -23500.418,E2 -23500.418} C_VEL
LIN {X 0,Y 157.229,Z 394.979,A -85,B 0,C 180,E1 -23505.556,E2 -23505.556} C_VEL
LIN {X 0,Y 158.545,Z 393.954,A -85,B 0,C 180,E1 -23508.076,E2 -23508.076} C_VEL
LIN {X 0,Y 160.304,Z 392.547,A -85,B 0,C 180,E1 -23510.531,E2 -23510.531} C_VEL
LIN {X 0,Y 163.526,Z 389.642,A -85,B 0,C 180,E1 -23514.097,E2 -23514.097} C_VEL
LIN {X 0,Y 167.228,Z 385.792,A -85,B 0,C 180,E1 -23517.534,E2 -23517.534} C_VEL
LIN {X 0,Y 171.487,Z 380.892,A -85,B 0,C 180,E1 -23520.815,E2 -23520.815} C_VEL
LIN {X 0,Y 177.357,Z 373.648,A -85,B 0,C 180,E1 -23524.379,E2 -23524.379} C_VEL
LIN {X 0,Y 181.98,Z 367.256,A -85,B 0,C 180,E1 -23526.769,E2 -23526.769} C_VEL
LIN {X 0,Y 188.084,Z 357.975,A -85,B 0,C 180,E1 -23529.436,E2 -23529.436} C_VEL
LIN {X 0,Y 193.986,Z 347.507,A -85,B 0,C 180,E1 -23531.736,E2 -23531.736} C_VEL
LIN {X 0,Y 199.073,Z 336.918,A -85,B 0,C 180,E1 -23533.504,E2 -23533.504} C_VEL
LIN {X 0,Y 203.922,Z 325.035,A -85,B 0,C 180,E1 -23534.951,E2 -23534.951} C_VEL
LIN {X 0,Y 207.656,Z 313.728,A -85,B 0,C 180,E1 -23535.987,E2 -23535.987} C_VEL
LIN {X 0,Y 210.956,Z 300.587,A -85,B 0,C 180,E1 -23536.869,E2 -23536.869} C_VEL
LIN {X 0,Y 213.38,Z 286.214,A -85,B 0,C 180,E1 -23537.507,E2 -23537.507} C_VEL
LIN {X 0,Y 215.96,Z 262.719,A -85,B 0,C 180,E1 -23538.387,E2 -23538.387} C_VEL
LIN {X 0,Y 213.546,Z 255.837,A -85,B 0,C 180,E1 -23540.528,E2 -23540.528} C_VEL
LIN {X 0,Y 210.959,Z 249.317,A -85,B 0,C 180,E1 -23543.153,E2 -23543.153} C_VEL
LIN {X 0,Y 209.068,Z 245.223,A -85,B 0,C 180,E1 -23545.328,E2 -23545.328} C_VEL
LIN {X 0,Y 207.263,Z 241.039,A -85,B 0,C 180,E1 -23548.045,E2 -23548.045} C_VEL
LIN {X 0,Y 205.062,Z 236.181,A -85,B 0,C 180,E1 -23553.248,E2 -23553.248} C_VEL
LIN {X 0,Y 204.552,Z 235.246,A -85,B 0,C 180,E1 -23556.935,E2 -23556.935} C_VEL
LIN {X 0,Y 205.262,Z 235.446,A -85,B 0,C 180,E1 -23561.491,E2 -23561.491} C_VEL
LIN {X 0,Y 208.083,Z 239.855,A -85,B 0,C 180,E1 -23567.199,E2 -23567.199} C_VEL
LIN {X 0,Y 210.174,Z 243.813,A -85,B 0,C 180,E1 -23569.962,E2 -23569.962} C_VEL
LIN {X 0,Y 212.402,Z 247.708,A -85,B 0,C 180,E1 -23572.241,E2 -23572.241} C_VEL
LIN {X 0,Y 215.867,Z 255.837,A -85,B 0,C 180,E1 -23575.374,E2 -23575.374} C_VEL
LIN {X 0,Y 216.503,Z 257.473,A -85,B 0,C 180,E1 -23575.901,E2 -23575.901} C_VEL
LIN {X 0,Y 212.847,Z 287.795,A -85,B 0,C 180,E1 -23577.001,E2 -23577.001} C_VEL
LIN {X 0,Y 210.138,Z 301.305,A -85,B 0,C 180,E1 -23577.769,E2 -23577.769} C_VEL
LIN {X 0,Y 206.436,Z 314.566,A -85,B 0,C 180,E1 -23578.902,E2 -23578.902} C_VEL
LIN {X 0,Y 202.376,Z 326.059,A -85,B 0,C 180,E1 -23580.248,E2 -23580.248} C_VEL
LIN {X 0,Y 197.25,Z 337.746,A -85,B 0,C 180,E1 -23582.041,E2 -23582.041} C_VEL
LIN {X 0,Y 191.641,Z 348.384,A -85,B 0,C 180,E1 -23584.205,E2 -23584.205} C_VEL
LIN {X 0,Y 186.298,Z 357.078,A -85,B 0,C 180,E1 -23586.497,E2 -23586.497} C_VEL
LIN {X 0,Y 181.307,Z 364.231,A -85,B 0,C 180,E1 -23588.919,E2 -23588.919} C_VEL
LIN {X 0,Y 175.871,Z 371.189,A -85,B 0,C 180,E1 -23591.974,E2 -23591.974} C_VEL
LIN {X 0,Y 170.678,Z 377.08,A -85,B 0,C 180,E1 -23595.47,E2 -23595.47} C_VEL
LIN {X 0,Y 165.376,Z 382.317,A -85,B 0,C 180,E1 -23599.874,E2 -23599.874} C_VEL
LIN {X 0,Y 161.578,Z 385.482,A -85,B 0,C 180,E1 -23604.021,E2 -23604.021} C_VEL
LIN {X 0,Y 158.906,Z 387.258,A -85,B 0,C 180,E1 -23607.807,E2 -23607.807} C_VEL
LIN {X 0,Y 156.46,Z 388.131,A -85,B 0,C 180,E1 -23612.616,E2 -23612.616} C_VEL
LIN {X 0,Y 155.274,Z 387.933,A -85,B 0,C 180,E1 -23616.042,E2 -23616.042} C_VEL
LIN {X 0,Y 154.57,Z 387,A -85,B 0,C 180,E1 -23619.534,E2 -23619.534} C_VEL
LIN {X 0,Y 154.253,Z 385.256,A -85,B 0,C 180,E1 -23623.2,E2 -23623.2} C_VEL
LIN {X 0,Y 154.384,Z 382.629,A -85,B 0,C 180,E1 -23626.935,E2 -23626.935} C_VEL
LIN {X 0,Y 155.04,Z 378.181,A -85,B 0,C 180,E1 -23631.444,E2 -23631.444} C_VEL
LIN {X 0,Y 156.103,Z 372.24,A -85,B 0,C 180,E1 -23635.893,E2 -23635.893} C_VEL
LIN {X 0,Y 157.65,Z 364.819,A -85,B 0,C 180,E1 -23640.102,E2 -23640.102} C_VEL
LIN {X 0,Y 159.596,Z 356.338,A -85,B 0,C 180,E1 -23643.874,E2 -23643.874} C_VEL
LIN {X 0,Y 162.048,Z 346.24,A -85,B 0,C 180,E1 -23647.363,E2 -23647.363} C_VEL
LIN {X 0,Y 164.536,Z 335.32,A -85,B 0,C 180,E1 -23650.325,E2 -23650.325} C_VEL
LIN {X 0,Y 166.65,Z 325.046,A -85,B 0,C 180,E1 -23652.514,E2 -23652.514} C_VEL
LIN {X 0,Y 168.883,Z 312.581,A -85,B 0,C 180,E1 -23654.568,E2 -23654.568} C_VEL
LIN {X 0,Y 170.668,Z 300.478,A -85,B 0,C 180,E1 -23656.063,E2 -23656.063} C_VEL
LIN {X 0,Y 172.088,Z 287.234,A -85,B 0,C 180,E1 -23657.206,E2 -23657.206} C_VEL
LIN {X 0,Y 173.254,Z 270.409,A -85,B 0,C 180,E1 -23658.098,E2 -23658.098} C_VEL
LIN {X 0,Y 175.931,Z 227.786,A -85,B 0,C 180,E1 -23660.054,E2 -23660.054} C_VEL
LIN {X 0,Y 170.393,Z 211.538,A -85,B 0,C 180,E1 -23661.843,E2 -23661.843} C_VEL
LIN {X 0,Y 162.232,Z 193.323,A -85,B 0,C 180,E1 -23664.395,E2 -23664.395} C_VEL
LIN {X 0,Y 157.883,Z 184.669,A -85,B 0,C 180,E1 -23665.812,E2 -23665.812} C_VEL
LIN {X 0,Y 157.746,Z 183.838,A -85,B 0,C 180,E1 -23666.009,E2 -23666.009} C_VEL
LIN {X 0,Y 158.233,Z 183.78,A -85,B 0,C 180,E1 -23670,E2 -23670} C_VEL
LIN {X 0,Y 157.755,Z 183.838,A -85,B 0,C 180,E1 -23677.681,E2 -23677.681} C_VEL
LIN {X 0,Y 157.628,Z 183.853,A -85,B 0,C 180,E1 -23681.224,E2 -23681.224} C_VEL
LIN {X 0,Y 157.403,Z 183.881,A -85,B 0,C 180,E1 -23685.539,E2 -23685.539} C_VEL
LIN {X 0,Y 157.299,Z 183.888,A -85,B 0,C 180,E1 -23690.943,E2 -23690.943} C_VEL
LIN {X 0,Y 157.263,Z 183.895,A -85,B 0,C 180,E1 -23696.65,E2 -23696.65} C_VEL
LIN {X 0,Y 157.261,Z 183.881,A -85,B 0,C 180,E1 -23702.431,E2 -23702.431} C_VEL
LIN {X 0,Y 157.255,Z 183.895,A -85,B 0,C 180,E1 -23706.445,E2 -23706.445} C_VEL
LIN {X 0,Y 157.186,Z 183.889,A -85,B 0,C 180,E1 -23712.119,E2 -23712.119} C_VEL
LIN {X 0,Y 157.186,Z 183.902,A -85,B 0,C 180,E1 -23717.883,E2 -23717.883} C_VEL
LIN {X 0,Y 157.256,Z 183.886,A -85,B 0,C 180,E1 -23723.557,E2 -23723.557} C_VEL
LIN {X 0,Y 157.277,Z 183.874,A -85,B 0,C 180,E1 -23728.105,E2 -23728.105} C_VEL
LIN {X 0,Y 157.264,Z 183.894,A -85,B 0,C 180,E1 -23733.457,E2 -23733.457} C_VEL
LIN {X 0,Y 157.357,Z 183.865,A -85,B 0,C 180,E1 -23739.704,E2 -23739.704} C_VEL
LIN {X 0,Y 157.402,Z 183.865,A -85,B 0,C 180,E1 -23744.462,E2 -23744.462} C_VEL
LIN {X 0,Y 157.683,Z 183.839,A -85,B 0,C 180,E1 -23749.731,E2 -23749.731} C_VEL
LIN {X 0,Y 157.752,Z 183.822,A -85,B 0,C 180,E1 -23752.32,E2 -23752.32} C_VEL
LIN {X 0,Y 158.233,Z 183.771,A -85,B 0,C 180,E1 -23760.001,E2 -23760.001} C_VEL
LIN {X 0,Y 157.753,Z 183.818,A -85,B 0,C 180,E1 -23767.682,E2 -23767.682} C_VEL
LIN {X 0,Y 157.629,Z 183.848,A -85,B 0,C 180,E1 -23771.223,E2 -23771.223} C_VEL
LIN {X 0,Y 157.401,Z 183.87,A -85,B 0,C 180,E1 -23775.541,E2 -23775.541} C_VEL
LIN {X 0,Y 157.302,Z 183.891,A -85,B 0,C 180,E1 -23780.943,E2 -23780.943} C_VEL
LIN {X 0,Y 157.267,Z 183.896,A -85,B 0,C 180,E1 -23786.65,E2 -23786.65} C_VEL
LIN {X 0,Y 157.261,Z 183.878,A -85,B 0,C 180,E1 -23792.432,E2 -23792.432} C_VEL
LIN {X 0,Y 157.259,Z 183.892,A -85,B 0,C 180,E1 -23796.445,E2 -23796.445} C_VEL
LIN {X 0,Y 157.19,Z 183.905,A -85,B 0,C 180,E1 -23802.119,E2 -23802.119} C_VEL
LIN {X 0,Y 157.229,Z 183.937,A -85,B 0,C 180,E1 -23807.188,E2 -23807.188} C_VEL
LIN {X 0,Y 157.444,Z 184.823,A -85,B 0,C 180,E1 -23807.622,E2 -23807.622} C_VEL
LIN {X 0,Y 165.494,Z 204.029,A -85,B 0,C 180,E1 -23810.383,E2 -23810.383} C_VEL
LIN {X 0,Y 171.492,Z 220.863,A -85,B 0,C 180,E1 -23812.392,E2 -23812.392} C_VEL
LIN {X 0,Y 173.752,Z 228.226,A -85,B 0,C 180,E1 -23813.161,E2 -23813.161} C_VEL
LIN {X 0,Y 175.245,Z 243.526,A -85,B 0,C 180,E1 -23814.231,E2 -23814.231} C_VEL
LIN {X 0,Y 172.116,Z 293.915,A -85,B 0,C 180,E1 -23816.635,E2 -23816.635} C_VEL
LIN {X 0,Y 170.656,Z 307.399,A -85,B 0,C 180,E1 -23817.718,E2 -23817.718} C_VEL
LIN {X 0,Y 168.834,Z 319.831,A -85,B 0,C 180,E1 -23819.168,E2 -23819.168} C_VEL
LIN {X 0,Y 166.267,Z 332.942,A -85,B 0,C 180,E1 -23821.261,E2 -23821.261} C_VEL
LIN {X 0,Y 163.887,Z 343.977,A -85,B 0,C 180,E1 -23823.582,E2 -23823.582} C_VEL
LIN {X 0,Y 161.388,Z 354.709,A -85,B 0,C 180,E1 -23826.5,E2 -23826.5} C_VEL
LIN {X 0,Y 159.119,Z 364.744,A -85,B 0,C 180,E1 -23829.983,E2 -23829.983} C_VEL
LIN {X 0,Y 157.181,Z 373.228,A -85,B 0,C 180,E1 -23833.772,E2 -23833.772} C_VEL
LIN {X 0,Y 155.884,Z 380.041,A -85,B 0,C 180,E1 -23837.634,E2 -23837.634} C_VEL
LIN {X 0,Y 155.601,Z 381.869,A -85,B 0,C 180,E1 -23838.852,E2 -23838.852} C_VEL
LIN {X 0,Y 154.561,Z 384.477,A -85,B 0,C 180,E1 -23840.782,E2 -23840.782} C_VEL
LIN {X 0,Y 151.313,Z 388.013,A -85,B 0,C 180,E1 -23844.044,E2 -23844.044} C_VEL
LIN {X 0,Y 148.814,Z 390.316,A -85,B 0,C 180,E1 -23846.813,E2 -23846.813} C_VEL
LIN {X 0,Y 147.87,Z 391.846,A -85,B 0,C 180,E1 -23849.005,E2 -23849.005} C_VEL
LIN {X 0,Y 147.849,Z 392.308,A -85,B 0,C 180,E1 -23849.748,E2 -23849.748} C_VEL
LIN {X 0,Y 147.718,Z 393.897,A -85,B 0,C 180,E1 -23852.727,E2 -23852.727} C_VEL
LIN {X 0,Y 147.944,Z 395.458,A -85,B 0,C 180,E1 -23858.193,E2 -23858.193} C_VEL
LIN {X 0,Y 149.262,Z 395.515,A -85,B 0,C 180,E1 -23863.616,E2 -23863.616} C_VEL
LIN {X 0,Y 151.798,Z 394.016,A -85,B 0,C 180,E1 -23868.91,E2 -23868.91} C_VEL
LIN {X 0,Y 155.863,Z 390.992,A -85,B 0,C 180,E1 -23873.941,E2 -23873.941} C_VEL
LIN {X 0,Y 159.712,Z 387.623,A -85,B 0,C 180,E1 -23877.518,E2 -23877.518} C_VEL
LIN {X 0,Y 163.839,Z 383.274,A -85,B 0,C 180,E1 -23880.98,E2 -23880.98} C_VEL
LIN {X 0,Y 168.913,Z 377.792,A -85,B 0,C 180,E1 -23884.172,E2 -23884.172} C_VEL
LIN {X 0,Y 174.367,Z 371.085,A -85,B 0,C 180,E1 -23887.198,E2 -23887.198} C_VEL
LIN {X 0,Y 180.621,Z 362.771,A -85,B 0,C 180,E1 -23889.941,E2 -23889.941} C_VEL
LIN {X 0,Y 187.192,Z 352.452,A -85,B 0,C 180,E1 -23892.515,E2 -23892.515} C_VEL
LIN {X 0,Y 192.914,Z 341.871,A -85,B 0,C 180,E1 -23894.529,E2 -23894.529} C_VEL
LIN {X 0,Y 197.849,Z 331.38,A -85,B 0,C 180,E1 -23895.997,E2 -23895.997} C_VEL
LIN {X 0,Y 202.273,Z 319.963,A -85,B 0,C 180,E1 -23897.22,E2 -23897.22} C_VEL
LIN {X 0,Y 206.198,Z 307.268,A -85,B 0,C 180,E1 -23898.208,E2 -23898.208} C_VEL
LIN {X 0,Y 209.144,Z 293.927,A -85,B 0,C 180,E1 -23898.931,E2 -23898.931} C_VEL
LIN {X 0,Y 211.858,Z 272.966,A -85,B 0,C 180,E1 -23899.726,E2 -23899.726} C_VEL
LIN {X 0,Y 212.616,Z 265.891,A -85,B 0,C 180,E1 -23900.018,E2 -23900.018} C_VEL
LIN {X 0,Y 210.203,Z 258.849,A -85,B 0,C 180,E1 -23902.484,E2 -23902.484} C_VEL
LIN {X 0,Y 208.319,Z 254.079,A -85,B 0,C 180,E1 -23904.659,E2 -23904.659} C_VEL
LIN {X 0,Y 207.115,Z 251.189,A -85,B 0,C 180,E1 -23906.306,E2 -23906.306} C_VEL
LIN {X 0,Y 205.673,Z 247.635,A -85,B 0,C 180,E1 -23908.677,E2 -23908.677} C_VEL
LIN {X 0,Y 203.89,Z 243.206,A -85,B 0,C 180,E1 -23913.377,E2 -23913.377} C_VEL
LIN {X 0,Y 203.432,Z 242.26,A -85,B 0,C 180,E1 -23916.8,E2 -23916.8} C_VEL
LIN {X 0,Y 204.091,Z 242.454,A -85,B 0,C 180,E1 -23921.381,E2 -23921.381} C_VEL
LIN {X 0,Y 206.55,Z 246.593,A -85,B 0,C 180,E1 -23926.711,E2 -23926.711} C_VEL
LIN {X 0,Y 208.298,Z 250.106,A -85,B 0,C 180,E1 -23929.222,E2 -23929.222} C_VEL
LIN {X 0,Y 210.5,Z 254.236,A -85,B 0,C 180,E1 -23931.647,E2 -23931.647} C_VEL
LIN {X 0,Y 213.119,Z 261.018,A -85,B 0,C 180,E1 -23934.277,E2 -23934.277} C_VEL
LIN {X 0,Y 209.842,Z 287.52,A -85,B 0,C 180,E1 -23935.243,E2 -23935.243} C_VEL
LIN {X 0,Y 207.127,Z 300.874,A -85,B 0,C 180,E1 -23935.988,E2 -23935.988} C_VEL
LIN {X 0,Y 203.768,Z 312.828,A -85,B 0,C 180,E1 -23936.949,E2 -23936.949} C_VEL
LIN {X 0,Y 199.761,Z 323.981,A -85,B 0,C 180,E1 -23938.173,E2 -23938.173} C_VEL
LIN {X 0,Y 195.147,Z 334.533,A -85,B 0,C 180,E1 -23939.688,E2 -23939.688} C_VEL
LIN {X 0,Y 189.328,Z 345.612,A -85,B 0,C 180,E1 -23941.725,E2 -23941.725} C_VEL
LIN {X 0,Y 183.211,Z 355.494,A -85,B 0,C 180,E1 -23944.176,E2 -23944.176} C_VEL
LIN {X 0,Y 177.299,Z 363.687,A -85,B 0,C 180,E1 -23946.829,E2 -23946.829} C_VEL
LIN {X 0,Y 171.268,Z 371.02,A -85,B 0,C 180,E1 -23949.996,E2 -23949.996} C_VEL
LIN {X 0,Y 166.055,Z 376.577,A -85,B 0,C 180,E1 -23953.242,E2 -23953.242} C_VEL
LIN {X 0,Y 161.415,Z 380.974,A -85,B 0,C 180,E1 -23956.693,E2 -23956.693} C_VEL
LIN {X 0,Y 156.809,Z 384.742,A -85,B 0,C 180,E1 -23961.01,E2 -23961.01} C_VEL
LIN {X 0,Y 154.08,Z 386.617,A -85,B 0,C 180,E1 -23964.236,E2 -23964.236} C_VEL
LIN {X 0,Y 151.441,Z 387.948,A -85,B 0,C 180,E1 -23968.149,E2 -23968.149} C_VEL
LIN {X 0,Y 149.476,Z 388.371,A -85,B 0,C 180,E1 -23972.189,E2 -23972.189} C_VEL
LIN {X 0,Y 148.091,Z 387.909,A -85,B 0,C 180,E1 -23976.22,E2 -23976.22} C_VEL
LIN {X 0,Y 147.2,Z 385.792,A -85,B 0,C 180,E1 -23981.944,E2 -23981.944} C_VEL
LIN {X 0,Y 147.194,Z 383.415,A -85,B 0,C 180,E1 -23985.74,E2 -23985.74} C_VEL
LIN {X 0,Y 147.605,Z 380.064,A -85,B 0,C 180,E1 -23989.623,E2 -23989.623} C_VEL
LIN {X 0,Y 148.386,Z 375.549,A -85,B 0,C 180,E1 -23993.625,E2 -23993.625} C_VEL
LIN {X 0,Y 149.573,Z 369.561,A -85,B 0,C 180,E1 -23997.752,E2 -23997.752} C_VEL
LIN {X 0,Y 151.298,Z 361.71,A -85,B 0,C 180,E1 -24001.952,E2 -24001.952} C_VEL
LIN {X 0,Y 153.487,Z 352.898,A -85,B 0,C 180,E1 -24005.664,E2 -24005.664} C_VEL
LIN {X 0,Y 155.856,Z 343.294,A -85,B 0,C 180,E1 -24008.855,E2 -24008.855} C_VEL
LIN {X 0,Y 158.551,Z 331.458,A -85,B 0,C 180,E1 -24011.924,E2 -24011.924} C_VEL
LIN {X 0,Y 160.745,Z 320.552,A -85,B 0,C 180,E1 -24014.123,E2 -24014.123} C_VEL
LIN {X 0,Y 163.08,Z 307.255,A -85,B 0,C 180,E1 -24016.131,E2 -24016.131} C_VEL
LIN {X 0,Y 164.754,Z 294.185,A -85,B 0,C 180,E1 -24017.568,E2 -24017.568} C_VEL
LIN {X 0,Y 166.143,Z 279.913,A -85,B 0,C 180,E1 -24018.559,E2 -24018.559} C_VEL
LIN {X 0,Y 169.317,Z 228.835,A -85,B 0,C 180,E1 -24021.021,E2 -24021.021} C_VEL
LIN {X 0,Y 164.092,Z 213.712,A -85,B 0,C 180,E1 -24022.81,E2 -24022.81} C_VEL
LIN {X 0,Y 156.82,Z 197.284,A -85,B 0,C 180,E1 -24025.221,E2 -24025.221} C_VEL
LIN {X 0,Y 151.053,Z 185.711,A -85,B 0,C 180,E1 -24027.209,E2 -24027.209} C_VEL
LIN {X 0,Y 150.858,Z 184.695,A -85,B 0,C 180,E1 -24027.33,E2 -24027.33} C_VEL
LIN {X 0,Y 151.193,Z 184.657,A -85,B 0,C 180,E1 -24030,E2 -24030} C_VEL
LIN {X 0,Y 150.694,Z 184.72,A -85,B 0,C 180,E1 -24038.043,E2 -24038.043} C_VEL
LIN {X 0,Y 150.57,Z 184.733,A -85,B 0,C 180,E1 -24041.429,E2 -24041.429} C_VEL
LIN {X 0,Y 150.308,Z 184.76,A -85,B 0,C 180,E1 -24046.293,E2 -24046.293} C_VEL
LIN {X 0,Y 150.279,Z 184.762,A -85,B 0,C 180,E1 -24050.722,E2 -24050.722} C_VEL
LIN {X 0,Y 150.182,Z 184.778,A -85,B 0,C 180,E1 -24057.238,E2 -24057.238} C_VEL
LIN {X 0,Y 150.202,Z 184.761,A -85,B 0,C 180,E1 -24062.626,E2 -24062.626} C_VEL
LIN {X 0,Y 150.166,Z 184.78,A -85,B 0,C 180,E1 -24067.475,E2 -24067.475} C_VEL
LIN {X 0,Y 150.129,Z 184.77,A -85,B 0,C 180,E1 -24071.497,E2 -24071.497} C_VEL
LIN {X 0,Y 150.123,Z 184.772,A -85,B 0,C 180,E1 -24075.396,E2 -24075.396} C_VEL
LIN {X 0,Y 150.134,Z 184.784,A -85,B 0,C 180,E1 -24079.054,E2 -24079.054} C_VEL
LIN {X 0,Y 150.173,Z 184.772,A -85,B 0,C 180,E1 -24082.711,E2 -24082.711} C_VEL
LIN {X 0,Y 150.202,Z 184.751,A -85,B 0,C 180,E1 -24087.375,E2 -24087.375} C_VEL
LIN {X 0,Y 150.182,Z 184.777,A -85,B 0,C 180,E1 -24092.764,E2 -24092.764} C_VEL
LIN {X 0,Y 150.279,Z 184.749,A -85,B 0,C 180,E1 -24099.28,E2 -24099.28} C_VEL
LIN {X 0,Y 150.308,Z 184.745,A -85,B 0,C 180,E1 -24103.709,E2 -24103.709} C_VEL
LIN {X 0,Y 150.603,Z 184.721,A -85,B 0,C 180,E1 -24109.243,E2 -24109.243} C_VEL
LIN {X 0,Y 150.675,Z 184.705,A -85,B 0,C 180,E1 -24111.957,E2 -24111.957} C_VEL
LIN {X 0,Y 151.193,Z 184.648,A -85,B 0,C 180,E1 -24120.001,E2 -24120.001} C_VEL
LIN {X 0,Y 150.676,Z 184.701,A -85,B 0,C 180,E1 -24128.045,E2 -24128.045} C_VEL
LIN {X 0,Y 150.572,Z 184.728,A -85,B 0,C 180,E1 -24131.427,E2 -24131.427} C_VEL
LIN {X 0,Y 150.307,Z 184.75,A -85,B 0,C 180,E1 -24136.294,E2 -24136.294} C_VEL
LIN {X 0,Y 150.281,Z 184.766,A -85,B 0,C 180,E1 -24140.722,E2 -24140.722} C_VEL
LIN {X 0,Y 150.183,Z 184.78,A -85,B 0,C 180,E1 -24147.236,E2 -24147.236} C_VEL
LIN {X 0,Y 150.202,Z 184.755,A -85,B 0,C 180,E1 -24152.625,E2 -24152.625} C_VEL
LIN {X 0,Y 150.17,Z 184.78,A -85,B 0,C 180,E1 -24157.476,E2 -24157.476} C_VEL
LIN {X 0,Y 150.134,Z 184.786,A -85,B 0,C 180,E1 -24161.498,E2 -24161.498} C_VEL
LIN {X 0,Y 150.173,Z 184.778,A -85,B 0,C 180,E1 -24166.005,E2 -24166.005} C_VEL
LIN {X 0,Y 151.216,Z 187.646,A -85,B 0,C 180,E1 -24166.481,E2 -24166.481} C_VEL
LIN {X 0,Y 153.777,Z 192.914,A -85,B 0,C 180,E1 -24167.388,E2 -24167.388} C_VEL
LIN {X 0,Y 160.021,Z 208.101,A -85,B 0,C 180,E1 -24169.613,E2 -24169.613} C_VEL
LIN {X 0,Y 166.853,Z 227.93,A -85,B 0,C 180,E1 -24172.043,E2 -24172.043} C_VEL
LIN {X 0,Y 167.662,Z 232.123,A -85,B 0,C 180,E1 -24172.422,E2 -24172.422} C_VEL
LIN {X 0,Y 168.737,Z 244.057,A -85,B 0,C 180,E1 -24173.283,E2 -24173.283} C_VEL
LIN {X 0,Y 165.599,Z 293.02,A -85,B 0,C 180,E1 -24175.691,E2 -24175.691} C_VEL
LIN {X 0,Y 164.091,Z 306.703,A -85,B 0,C 180,E1 -24176.81,E2 -24176.81} C_VEL
LIN {X 0,Y 162.2,Z 319.276,A -85,B 0,C 180,E1 -24178.307,E2 -24178.307} C_VEL
LIN {X 0,Y 159.711,Z 331.684,A -85,B 0,C 180,E1 -24180.327,E2 -24180.327} C_VEL
LIN {X 0,Y 157.237,Z 342.922,A -85,B 0,C 180,E1 -24182.733,E2 -24182.733} C_VEL
LIN {X 0,Y 154.97,Z 352.479,A -85,B 0,C 180,E1 -24185.33,E2 -24185.33} C_VEL
LIN {X 0,Y 152.806,Z 361.507,A -85,B 0,C 180,E1 -24188.411,E2 -24188.411} C_VEL
LIN {X 0,Y 150.691,Z 370.639,A -85,B 0,C 180,E1 -24192.353,E2 -24192.353} C_VEL
LIN {X 0,Y 149.124,Z 377.95,A -85,B 0,C 180,E1 -24196.37,E2 -24196.37} C_VEL
LIN {X 0,Y 148.224,Z 383.74,A -85,B 0,C 180,E1 -24200.447,E2 -24200.447} C_VEL
LIN {X 0,Y 147.823,Z 388.248,A -85,B 0,C 180,E1 -24204.543,E2 -24204.543} C_VEL
LIN {X 0,Y 147.758,Z 390.592,A -85,B 0,C 180,E1 -24207.273,E2 -24207.273} C_VEL
LIN {X 0,Y 147.849,Z 392.308,A -85,B 0,C 180,E1 -24209.748,E2 -24209.748} C_VEL
LIN {X 0,Y 147.625,Z 393.231,A -85,B 0,C 180,E1 -24211.222,E2 -24211.222} C_VEL
LIN {X 0,Y 146.845,Z 393.965,A -85,B 0,C 180,E1 -24212.694,E2 -24212.694} C_VEL
LIN {X 0,Y 144.448,Z 394.933,A -85,B 0,C 180,E1 -24215.651,E2 -24215.651} C_VEL
LIN {X 0,Y 142.166,Z 395.367,A -85,B 0,C 180,E1 -24218.74,E2 -24218.74} C_VEL
LIN {X 0,Y 141.492,Z 395.436,A -85,B 0,C 180,E1 -24221.148,E2 -24221.148} C_VEL
LIN {X 0,Y 141.602,Z 395.421,A -85,B 0,C 180,E1 -24221.956,E2 -24221.956} C_VEL
LIN {X 0,Y 143.527,Z 394.907,A -85,B 0,C 180,E1 -24227.085,E2 -24227.085} C_VEL
LIN {X 0,Y 145.09,Z 394.09,A -85,B 0,C 180,E1 -24229.82,E2 -24229.82} C_VEL
LIN {X 0,Y 149.395,Z 391.237,A -85,B 0,C 180,E1 -24235.048,E2 -24235.048} C_VEL
LIN {X 0,Y 154.774,Z 386.806,A -85,B 0,C 180,E1 -24239.965,E2 -24239.965} C_VEL
LIN {X 0,Y 159.526,Z 382.309,A -85,B 0,C 180,E1 -24243.414,E2 -24243.414} C_VEL
LIN {X 0,Y 165.957,Z 375.591,A -85,B 0,C 180,E1 -24247.117,E2 -24247.117} C_VEL
LIN {X 0,Y 170.957,Z 369.714,A -85,B 0,C 180,E1 -24249.582,E2 -24249.582} C_VEL
LIN {X 0,Y 177.539,Z 361.114,A -85,B 0,C 180,E1 -24252.294,E2 -24252.294} C_VEL
LIN {X 0,Y 184.49,Z 350.589,A -85,B 0,C 180,E1 -24254.808,E2 -24254.808} C_VEL
LIN {X 0,Y 189.936,Z 340.821,A -85,B 0,C 180,E1 -24256.564,E2 -24256.564} C_VEL
LIN {X 0,Y 195.721,Z 328.633,A -85,B 0,C 180,E1 -24258.166,E2 -24258.166} C_VEL
LIN {X 0,Y 200.321,Z 316.553,A -85,B 0,C 180,E1 -24259.347,E2 -24259.347} C_VEL
LIN {X 0,Y 204.353,Z 302.641,A -85,B 0,C 180,E1 -24260.298,E2 -24260.298} C_VEL
LIN {X 0,Y 207.056,Z 289.182,A -85,B 0,C 180,E1 -24260.92,E2 -24260.92} C_VEL
LIN {X 0,Y 209.494,Z 269.453,A -85,B 0,C 180,E1 -24261.669,E2 -24261.669} C_VEL
LIN {X 0,Y 207.597,Z 263.566,A -85,B 0,C 180,E1 -24263.911,E2 -24263.911} C_VEL
LIN {X 0,Y 205.865,Z 258.587,A -85,B 0,C 180,E1 -24266.323,E2 -24266.323} C_VEL
LIN {X 0,Y 204.149,Z 254.252,A -85,B 0,C 180,E1 -24269.275,E2 -24269.275} C_VEL
LIN {X 0,Y 202.669,Z 250.075,A -85,B 0,C 180,E1 -24273.766,E2 -24273.766} C_VEL
LIN {X 0,Y 202.288,Z 249.217,A -85,B 0,C 180,E1 -24277.531,E2 -24277.531} C_VEL
LIN {X 0,Y 202.915,Z 249.492,A -85,B 0,C 180,E1 -24281.269,E2 -24281.269} C_VEL
LIN {X 0,Y 205.046,Z 253.337,A -85,B 0,C 180,E1 -24286.241,E2 -24286.241} C_VEL
LIN {X 0,Y 206.846,Z 257.205,A -85,B 0,C 180,E1 -24288.96,E2 -24288.96} C_VEL
LIN {X 0,Y 208.485,Z 260.486,A -85,B 0,C 180,E1 -24290.897,E2 -24290.897} C_VEL
LIN {X 0,Y 209.991,Z 265.063,A -85,B 0,C 180,E1 -24292.65,E2 -24292.65} C_VEL
LIN {X 0,Y 206.798,Z 288.81,A -85,B 0,C 180,E1 -24293.503,E2 -24293.503} C_VEL
LIN {X 0,Y 204.126,Z 301.201,A -85,B 0,C 180,E1 -24294.194,E2 -24294.194} C_VEL
LIN {X 0,Y 200.742,Z 312.829,A -85,B 0,C 180,E1 -24295.104,E2 -24295.104} C_VEL
LIN {X 0,Y 196.255,Z 324.829,A -85,B 0,C 180,E1 -24296.405,E2 -24296.405} C_VEL
LIN {X 0,Y 191.468,Z 335.269,A -85,B 0,C 180,E1 -24297.896,E2 -24297.896} C_VEL
LIN {X 0,Y 185.812,Z 345.54,A -85,B 0,C 180,E1 -24299.767,E2 -24299.767} C_VEL
LIN {X 0,Y 180.233,Z 354.215,A -85,B 0,C 180,E1 -24301.836,E2 -24301.836} C_VEL
LIN {X 0,Y 173.483,Z 363.19,A -85,B 0,C 180,E1 -24304.646,E2 -24304.646} C_VEL
LIN {X 0,Y 167.139,Z 370.605,A -85,B 0,C 180,E1 -24307.776,E2 -24307.776} C_VEL
LIN {X 0,Y 161.065,Z 376.744,A -85,B 0,C 180,E1 -24311.323,E2 -24311.323} C_VEL
LIN {X 0,Y 156.787,Z 380.528,A -85,B 0,C 180,E1 -24314.27,E2 -24314.27} C_VEL
LIN {X 0,Y 153.949,Z 382.807,A -85,B 0,C 180,E1 -24316.532,E2 -24316.532} C_VEL
LIN {X 0,Y 149.937,Z 385.658,A -85,B 0,C 180,E1 -24320.374,E2 -24320.374} C_VEL
LIN {X 0,Y 145.665,Z 387.914,A -85,B 0,C 180,E1 -24325.735,E2 -24325.735} C_VEL
LIN {X 0,Y 143.563,Z 388.539,A -85,B 0,C 180,E1 -24329.309,E2 -24329.309} C_VEL
LIN {X 0,Y 141.967,Z 388.467,A -85,B 0,C 180,E1 -24332.992,E2 -24332.992} C_VEL
LIN {X 0,Y 140.782,Z 387.659,A -85,B 0,C 180,E1 -24336.992,E2 -24336.992} C_VEL
LIN {X 0,Y 140.168,Z 385.976,A -85,B 0,C 180,E1 -24341.229,E2 -24341.229} C_VEL
LIN {X 0,Y 140.084,Z 383.464,A -85,B 0,C 180,E1 -24345.383,E2 -24345.383} C_VEL
LIN {X 0,Y 140.48,Z 380.105,A -85,B 0,C 180,E1 -24349.432,E2 -24349.432} C_VEL
LIN {X 0,Y 141.411,Z 374.728,A -85,B 0,C 180,E1 -24354.271,E2 -24354.271} C_VEL
LIN {X 0,Y 142.814,Z 367.937,A -85,B 0,C 180,E1 -24358.92,E2 -24358.92} C_VEL
LIN {X 0,Y 144.342,Z 361.444,A -85,B 0,C 180,E1 -24362.449,E2 -24362.449} C_VEL
LIN {X 0,Y 146.562,Z 352.833,A -85,B 0,C 180,E1 -24366.219,E2 -24366.219} C_VEL
LIN {X 0,Y 149.078,Z 342.896,A -85,B 0,C 180,E1 -24369.634,E2 -24369.634} C_VEL
LIN {X 0,Y 151.567,Z 332.473,A -85,B 0,C 180,E1 -24372.459,E2 -24372.459} C_VEL
LIN {X 0,Y 154.045,Z 320.659,A -85,B 0,C 180,E1 -24374.961,E2 -24374.961} C_VEL
LIN {X 0,Y 156.412,Z 307.544,A -85,B 0,C 180,E1 -24377.018,E2 -24377.018} C_VEL
LIN {X 0,Y 158.122,Z 295.017,A -85,B 0,C 180,E1 -24378.457,E2 -24378.457} C_VEL
LIN {X 0,Y 159.527,Z 281.272,A -85,B 0,C 180,E1 -24379.476,E2 -24379.476} C_VEL
LIN {X 0,Y 162.884,Z 230.358,A -85,B 0,C 180,E1 -24382.017,E2 -24382.017} C_VEL
LIN {X 0,Y 158.352,Z 217.085,A -85,B 0,C 180,E1 -24383.665,E2 -24383.665} C_VEL
LIN {X 0,Y 151.127,Z 200.794,A -85,B 0,C 180,E1 -24386.167,E2 -24386.167} C_VEL
LIN {X 0,Y 144.106,Z 186.411,A -85,B 0,C 180,E1 -24388.777,E2 -24388.777} C_VEL
LIN {X 0,Y 143.986,Z 185.553,A -85,B 0,C 180,E1 -24388.951,E2 -24388.951} C_VEL
LIN {X 0,Y 144.152,Z 185.534,A -85,B 0,C 180,E1 -24390,E2 -24390} C_VEL
LIN {X 0,Y 143.616,Z 185.6,A -85,B 0,C 180,E1 -24398.442,E2 -24398.442} C_VEL
LIN {X 0,Y 143.495,Z 185.615,A -85,B 0,C 180,E1 -24401.614,E2 -24401.614} C_VEL
LIN {X 0,Y 143.248,Z 185.639,A -85,B 0,C 180,E1 -24407.12,E2 -24407.12} C_VEL
LIN {X 0,Y 143.215,Z 185.643,A -85,B 0,C 180,E1 -24411.194,E2 -24411.194} C_VEL
LIN {X 0,Y 143.139,Z 185.654,A -85,B 0,C 180,E1 -24417.9,E2 -24417.9} C_VEL
LIN {X 0,Y 143.133,Z 185.644,A -85,B 0,C 180,E1 -24423.415,E2 -24423.415} C_VEL
LIN {X 0,Y 143.049,Z 185.66,A -85,B 0,C 180,E1 -24429.694,E2 -24429.694} C_VEL
LIN {X 0,Y 143.03,Z 185.647,A -85,B 0,C 180,E1 -24433.465,E2 -24433.465} C_VEL
LIN {X 0,Y 143.034,Z 185.665,A -85,B 0,C 180,E1 -24437.478,E2 -24437.478} C_VEL
LIN {X 0,Y 143.069,Z 185.66,A -85,B 0,C 180,E1 -24441.81,E2 -24441.81} C_VEL
LIN {X 0,Y 143.17,Z 185.625,A -85,B 0,C 180,E1 -24447.32,E2 -24447.32} C_VEL
LIN {X 0,Y 143.103,Z 185.658,A -85,B 0,C 180,E1 -24453.77,E2 -24453.77} C_VEL
LIN {X 0,Y 143.243,Z 185.618,A -85,B 0,C 180,E1 -24459.914,E2 -24459.914} C_VEL
LIN {X 0,Y 143.301,Z 185.626,A -85,B 0,C 180,E1 -24465.807,E2 -24465.807} C_VEL
LIN {X 0,Y 143.53,Z 185.603,A -85,B 0,C 180,E1 -24468.706,E2 -24468.706} C_VEL
LIN {X 0,Y 143.602,Z 185.588,A -85,B 0,C 180,E1 -24471.558,E2 -24471.558} C_VEL
LIN {X 0,Y 144.152,Z 185.525,A -85,B 0,C 180,E1 -24480.001,E2 -24480.001} C_VEL
LIN {X 0,Y 143.603,Z 185.584,A -85,B 0,C 180,E1 -24488.444,E2 -24488.444} C_VEL
LIN {X 0,Y 143.496,Z 185.61,A -85,B 0,C 180,E1 -24491.613,E2 -24491.613} C_VEL
LIN {X 0,Y 143.248,Z 185.629,A -85,B 0,C 180,E1 -24497.121,E2 -24497.121} C_VEL
LIN {X 0,Y 143.218,Z 185.647,A -85,B 0,C 180,E1 -24501.194,E2 -24501.194} C_VEL
LIN {X 0,Y 143.139,Z 185.658,A -85,B 0,C 180,E1 -24507.898,E2 -24507.898} C_VEL
LIN {X 0,Y 143.134,Z 185.632,A -85,B 0,C 180,E1 -24513.414,E2 -24513.414} C_VEL
LIN {X 0,Y 143.053,Z 185.663,A -85,B 0,C 180,E1 -24519.694,E2 -24519.694} C_VEL
LIN {X 0,Y 143.083,Z 185.732,A -85,B 0,C 180,E1 -24524.423,E2 -24524.423} C_VEL
LIN {X 0,Y 144.12,Z 188.504,A -85,B 0,C 180,E1 -24524.877,E2 -24524.877} C_VEL
LIN {X 0,Y 147.693,Z 195.218,A -85,B 0,C 180,E1 -24526.208,E2 -24526.208} C_VEL
LIN {X 0,Y 153.835,Z 210.372,A -85,B 0,C 180,E1 -24528.551,E2 -24528.551} C_VEL
LIN {X 0,Y 159.44,Z 226.436,A -85,B 0,C 180,E1 -24530.645,E2 -24530.645} C_VEL
LIN {X 0,Y 161.19,Z 232.424,A -85,B 0,C 180,E1 -24531.334,E2 -24531.334} C_VEL
LIN {X 0,Y 162.29,Z 244.527,A -85,B 0,C 180,E1 -24532.262,E2 -24532.262} C_VEL
LIN {X 0,Y 159.015,Z 293.386,A -85,B 0,C 180,E1 -24534.761,E2 -24534.761} C_VEL
LIN {X 0,Y 157.392,Z 307.443,A -85,B 0,C 180,E1 -24535.975,E2 -24535.975} C_VEL
LIN {X 0,Y 155.417,Z 319.716,A -85,B 0,C 180,E1 -24537.521,E2 -24537.521} C_VEL
LIN {X 0,Y 152.88,Z 332.001,A -85,B 0,C 180,E1 -24539.624,E2 -24539.624} C_VEL
LIN {X 0,Y 150.308,Z 343.142,A -85,B 0,C 180,E1 -24542.123,E2 -24542.123} C_VEL
LIN {X 0,Y 148.073,Z 352.233,A -85,B 0,C 180,E1 -24544.712,E2 -24544.712} C_VEL
LIN {X 0,Y 145.758,Z 361.578,A -85,B 0,C 180,E1 -24548.057,E2 -24548.057} C_VEL
LIN {X 0,Y 143.566,Z 370.641,A -85,B 0,C 180,E1 -24552.184,E2 -24552.184} C_VEL
LIN {X 0,Y 141.999,Z 377.893,A -85,B 0,C 180,E1 -24556.403,E2 -24556.403} C_VEL
LIN {X 0,Y 141.227,Z 382.773,A -85,B 0,C 180,E1 -24559.969,E2 -24559.969} C_VEL
LIN {X 0,Y 140.773,Z 387.454,A -85,B 0,C 180,E1 -24564.269,E2 -24564.269} C_VEL
LIN {X 0,Y 140.701,Z 390.141,A -85,B 0,C 180,E1 -24567.459,E2 -24567.459} C_VEL
LIN {X 0,Y 140.799,Z 391.872,A -85,B 0,C 180,E1 -24570,E2 -24570} C_VEL
LIN {X 0,Y 140.649,Z 393.379,A -85,B 0,C 180,E1 -24572.864,E2 -24572.864} C_VEL
LIN {X 0,Y 140.632,Z 394.475,A -85,B 0,C 180,E1 -24575.736,E2 -24575.736} C_VEL
LIN {X 0,Y 141.476,Z 395.435,A -85,B 0,C 180,E1 -24581.461,E2 -24581.461} C_VEL
LIN {X 0,Y 141.602,Z 395.421,A -85,B 0,C 180,E1 -24581.956,E2 -24581.956} C_VEL
LIN {X 0,Y 141.688,Z 395.353,A -85,B 0,C 180,E1 -24584.346,E2 -24584.346} C_VEL
LIN {X 0,Y 140.608,Z 394.698,A -85,B 0,C 180,E1 -24588.343,E2 -24588.343} C_VEL
LIN {X 0,Y 140.266,Z 393.493,A -85,B 0,C 180,E1 -24592.348,E2 -24592.348} C_VEL
LIN {X 0,Y 141.475,Z 392.406,A -85,B 0,C 180,E1 -24594.651,E2 -24594.651} C_VEL
LIN {X 0,Y 145.74,Z 389.591,A -85,B 0,C 180,E1 -24598.83,E2 -24598.83} C_VEL
LIN {X 0,Y 151.901,Z 384.551,A -85,B 0,C 180,E1 -24603.724,E2 -24603.724} C_VEL
LIN {X 0,Y 157.482,Z 379.504,A -85,B 0,C 180,E1 -24607.046,E2 -24607.046} C_VEL
LIN {X 0,Y 164.498,Z 372.134,A -85,B 0,C 180,E1 -24610.657,E2 -24610.657} C_VEL
LIN {X 0,Y 171.314,Z 364.195,A -85,B 0,C 180,E1 -24613.404,E2 -24613.404} C_VEL
LIN {X 0,Y 178.43,Z 354.468,A -85,B 0,C 180,E1 -24615.957,E2 -24615.957} C_VEL
LIN {X 0,Y 184.589,Z 344.442,A -85,B 0,C 180,E1 -24617.938,E2 -24617.938} C_VEL
LIN {X 0,Y 190.51,Z 333.305,A -85,B 0,C 180,E1 -24619.539,E2 -24619.539} C_VEL
LIN {X 0,Y 195.239,Z 322.603,A -85,B 0,C 180,E1 -24620.707,E2 -24620.707} C_VEL
LIN {X 0,Y 199.418,Z 310.845,A -85,B 0,C 180,E1 -24621.654,E2 -24621.654} C_VEL
LIN {X 0,Y 202.872,Z 297.926,A -85,B 0,C 180,E1 -24622.39,E2 -24622.39} C_VEL
LIN {X 0,Y 205.262,Z 284.384,A -85,B 0,C 180,E1 -24622.942,E2 -24622.942} C_VEL
LIN {X 0,Y 206.626,Z 273.021,A -85,B 0,C 180,E1 -24623.393,E2 -24623.393} C_VEL
LIN {X 0,Y 204.929,Z 267.488,A -85,B 0,C 180,E1 -24625.748,E2 -24625.748} C_VEL
LIN {X 0,Y 203.629,Z 263.719,A -85,B 0,C 180,E1 -24627.901,E2 -24627.901} C_VEL
LIN {X 0,Y 202.622,Z 260.673,A -85,B 0,C 180,E1 -24630.046,E2 -24630.046} C_VEL
LIN {X 0,Y 201.44,Z 256.867,A -85,B 0,C 180,E1 -24634.279,E2 -24634.279} C_VEL
LIN {X 0,Y 201.144,Z 256.219,A -85,B 0,C 180,E1 -24637.396,E2 -24637.396} C_VEL
LIN {X 0,Y 201.742,Z 256.495,A -85,B 0,C 180,E1 -24641.156,E2 -24641.156} C_VEL
LIN {X 0,Y 203.522,Z 259.989,A -85,B 0,C 180,E1 -24645.704,E2 -24645.704} C_VEL
LIN {X 0,Y 205.158,Z 263.728,A -85,B 0,C 180,E1 -24648.341,E2 -24648.341} C_VEL
LIN {X 0,Y 206.514,Z 266.764,A -85,B 0,C 180,E1 -24650.147,E2 -24650.147} C_VEL
LIN {X 0,Y 207.133,Z 268.764,A -85,B 0,C 180,E1 -24650.942,E2 -24650.942} C_VEL
LIN {X 0,Y 204.132,Z 289.826,A -85,B 0,C 180,E1 -24651.689,E2 -24651.689} C_VEL
LIN {X 0,Y 201.137,Z 302.886,A -85,B 0,C 180,E1 -24652.418,E2 -24652.418} C_VEL
LIN {X 0,Y 196.921,Z 315.974,A -85,B 0,C 180,E1 -24653.489,E2 -24653.489} C_VEL
LIN {X 0,Y 191.826,Z 328.321,A -85,B 0,C 180,E1 -24654.895,E2 -24654.895} C_VEL
LIN {X 0,Y 185.674,Z 340.221,A -85,B 0,C 180,E1 -24656.744,E2 -24656.744} C_VEL
LIN {X 0,Y 179.953,Z 349.5,A -85,B 0,C 180,E1 -24658.6,E2 -24658.6} C_VEL
LIN {X 0,Y 174.54,Z 357.121,A -85,B 0,C 180,E1 -24660.575,E2 -24660.575} C_VEL
LIN {X 0,Y 168.125,Z 364.981,A -85,B 0,C 180,E1 -24663.181,E2 -24663.181} C_VEL
LIN {X 0,Y 160.995,Z 372.487,A -85,B 0,C 180,E1 -24666.605,E2 -24666.605} C_VEL
LIN {X 0,Y 154.344,Z 378.573,A -85,B 0,C 180,E1 -24670.493,E2 -24670.493} C_VEL
LIN {X 0,Y 149.902,Z 382.044,A -85,B 0,C 180,E1 -24673.556,E2 -24673.556} C_VEL
LIN {X 0,Y 146.016,Z 384.748,A -85,B 0,C 180,E1 -24676.784,E2 -24676.784} C_VEL
LIN {X 0,Y 142.439,Z 386.823,A -85,B 0,C 180,E1 -24680.373,E2 -24680.373} C_VEL
LIN {X 0,Y 139.104,Z 388.255,A -85,B 0,C 180,E1 -24684.578,E2 -24684.578} C_VEL
LIN {X 0,Y 136.518,Z 388.79,A -85,B 0,C 180,E1 -24688.938,E2 -24688.938} C_VEL
LIN {X 0,Y 134.656,Z 388.442,A -85,B 0,C 180,E1 -24693.378,E2 -24693.378} C_VEL
LIN {X 0,Y 133.251,Z 386.68,A -85,B 0,C 180,E1 -24699.264,E2 -24699.264} C_VEL
LIN {X 0,Y 133.003,Z 383.494,A -85,B 0,C 180,E1 -24704.997,E2 -24704.997} C_VEL
LIN {X 0,Y 133.373,Z 380.087,A -85,B 0,C 180,E1 -24709.276,E2 -24709.276} C_VEL
LIN {X 0,Y 134.085,Z 375.759,A -85,B 0,C 180,E1 -24713.445,E2 -24713.445} C_VEL
LIN {X 0,Y 135.235,Z 370.256,A -85,B 0,C 180,E1 -24717.644,E2 -24717.644} C_VEL
LIN {X 0,Y 136.837,Z 363.41,A -85,B 0,C 180,E1 -24721.806,E2 -24721.806} C_VEL
LIN {X 0,Y 139.203,Z 354.229,A -85,B 0,C 180,E1 -24726.179,E2 -24726.179} C_VEL
LIN {X 0,Y 141.694,Z 344.875,A -85,B 0,C 180,E1 -24729.685,E2 -24729.685} C_VEL
LIN {X 0,Y 144.187,Z 334.931,A -85,B 0,C 180,E1 -24732.63,E2 -24732.63} C_VEL
LIN {X 0,Y 146.711,Z 323.748,A -85,B 0,C 180,E1 -24735.228,E2 -24735.228} C_VEL
LIN {X 0,Y 148.888,Z 312.789,A -85,B 0,C 180,E1 -24737.205,E2 -24737.205} C_VEL
LIN {X 0,Y 151.012,Z 299.958,A -85,B 0,C 180,E1 -24738.931,E2 -24738.931} C_VEL
LIN {X 0,Y 152.529,Z 286.85,A -85,B 0,C 180,E1 -24740.151,E2 -24740.151} C_VEL
LIN {X 0,Y 154.482,Z 260.903,A -85,B 0,C 180,E1 -24741.586,E2 -24741.586} C_VEL
LIN {X 0,Y 156.489,Z 231.925,A -85,B 0,C 180,E1 -24743.068,E2 -24743.068} C_VEL
LIN {X 0,Y 152.42,Z 220.084,A -85,B 0,C 180,E1 -24744.611,E2 -24744.611} C_VEL
LIN {X 0,Y 145.658,Z 204.563,A -85,B 0,C 180,E1 -24747.124,E2 -24747.124} C_VEL
LIN {X 0,Y 137.928,Z 189.033,A -85,B 0,C 180,E1 -24750.165,E2 -24750.165} C_VEL
LIN {X 0,Y 136.974,Z 186.428,A -85,B 0,C 180,E1 -24750.735,E2 -24750.735} C_VEL
LIN {X 0,Y 136.543,Z 186.481,A -85,B 0,C 180,E1 -24758.883,E2 -24758.883} C_VEL
LIN {X 0,Y 136.41,Z 186.497,A -85,B 0,C 180,E1 -24761.893,E2 -24761.893} C_VEL
LIN {X 0,Y 136.161,Z 186.526,A -85,B 0,C 180,E1 -24768.041,E2 -24768.041} C_VEL
LIN {X 0,Y 136.14,Z 186.526,A -85,B 0,C 180,E1 -24771.69,E2 -24771.69} C_VEL
LIN {X 0,Y 136.058,Z 186.535,A -85,B 0,C 180,E1 -24778.586,E2 -24778.586} C_VEL
LIN {X 0,Y 136.036,Z 186.534,A -85,B 0,C 180,E1 -24784.631,E2 -24784.631} C_VEL
LIN {X 0,Y 136.021,Z 186.538,A -85,B 0,C 180,E1 -24789.195,E2 -24789.195} C_VEL
LIN {X 0,Y 135.975,Z 186.525,A -85,B 0,C 180,E1 -24793.649,E2 -24793.649} C_VEL
LIN {X 0,Y 135.979,Z 186.544,A -85,B 0,C 180,E1 -24797.788,E2 -24797.788} C_VEL
LIN {X 0,Y 136.018,Z 186.538,A -85,B 0,C 180,E1 -24801.683,E2 -24801.683} C_VEL
LIN {X 0,Y 136.049,Z 186.513,A -85,B 0,C 180,E1 -24805.743,E2 -24805.743} C_VEL
LIN {X 0,Y 136.083,Z 186.531,A -85,B 0,C 180,E1 -24812.304,E2 -24812.304} C_VEL
LIN {X 0,Y 136.178,Z 186.506,A -85,B 0,C 180,E1 -24818.824,E2 -24818.824} C_VEL
LIN {X 0,Y 136.22,Z 186.505,A -85,B 0,C 180,E1 -24825.052,E2 -24825.052} C_VEL
LIN {X 0,Y 136.424,Z 186.488,A -85,B 0,C 180,E1 -24828.18,E2 -24828.18} C_VEL
LIN {X 0,Y 136.531,Z 186.469,A -85,B 0,C 180,E1 -24831.118,E2 -24831.118} C_VEL
LIN {X 0,Y 137.109,Z 186.402,A -85,B 0,C 180,E1 -24840.001,E2 -24840.001} C_VEL
LIN {X 0,Y 136.532,Z 186.468,A -85,B 0,C 180,E1 -24848.885,E2 -24848.885} C_VEL
LIN {X 0,Y 136.413,Z 186.494,A -85,B 0,C 180,E1 -24851.894,E2 -24851.894} C_VEL
LIN {X 0,Y 136.161,Z 186.515,A -85,B 0,C 180,E1 -24858.042,E2 -24858.042} C_VEL
LIN {X 0,Y 136.142,Z 186.527,A -85,B 0,C 180,E1 -24861.69,E2 -24861.69} C_VEL
LIN {X 0,Y 136.059,Z 186.54,A -85,B 0,C 180,E1 -24868.584,E2 -24868.584} C_VEL
LIN {X 0,Y 136.039,Z 186.518,A -85,B 0,C 180,E1 -24874.632,E2 -24874.632} C_VEL
LIN {X 0,Y 136.025,Z 186.539,A -85,B 0,C 180,E1 -24879.195,E2 -24879.195} C_VEL
LIN {X 0,Y 136.025,Z 186.663,A -85,B 0,C 180,E1 -24882.648,E2 -24882.648} C_VEL
LIN {X 0,Y 136.978,Z 189.377,A -85,B 0,C 180,E1 -24883.117,E2 -24883.117} C_VEL
LIN {X 0,Y 138.327,Z 191.551,A -85,B 0,C 180,E1 -24883.644,E2 -24883.644} C_VEL
LIN {X 0,Y 142.241,Z 198.907,A -85,B 0,C 180,E1 -24885.177,E2 -24885.177} C_VEL
LIN {X 0,Y 148.361,Z 214.389,A -85,B 0,C 180,E1 -24887.684,E2 -24887.684} C_VEL
LIN {X 0,Y 153.826,Z 230.403,A -85,B 0,C 180,E1 -24889.854,E2 -24889.854} C_VEL
LIN {X 0,Y 154.971,Z 234.473,A -85,B 0,C 180,E1 -24890.33,E2 -24890.33} C_VEL
LIN {X 0,Y 155.86,Z 245.453,A -85,B 0,C 180,E1 -24891.189,E2 -24891.189} C_VEL
LIN {X 0,Y 152.52,Z 293.031,A -85,B 0,C 180,E1 -24893.713,E2 -24893.713} C_VEL
LIN {X 0,Y 150.925,Z 306.556,A -85,B 0,C 180,E1 -24894.914,E2 -24894.914} C_VEL
LIN {X 0,Y 148.865,Z 319.003,A -85,B 0,C 180,E1 -24896.511,E2 -24896.511} C_VEL
LIN {X 0,Y 146.076,Z 332.151,A -85,B 0,C 180,E1 -24898.855,E2 -24898.855} C_VEL
LIN {X 0,Y 143.339,Z 343.439,A -85,B 0,C 180,E1 -24901.522,E2 -24901.522} C_VEL
LIN {X 0,Y 140.575,Z 354.201,A -85,B 0,C 180,E1 -24904.852,E2 -24904.852} C_VEL
LIN {X 0,Y 138.298,Z 363.171,A -85,B 0,C 180,E1 -24908.381,E2 -24908.381} C_VEL
LIN {X 0,Y 136.442,Z 370.552,A -85,B 0,C 180,E1 -24911.998,E2 -24911.998} C_VEL
LIN {X 0,Y 134.863,Z 377.78,A -85,B 0,C 180,E1 -24916.437,E2 -24916.437} C_VEL
LIN {X 0,Y 133.999,Z 383.504,A -85,B 0,C 180,E1 -24920.947,E2 -24920.947} C_VEL
LIN {X 0,Y 133.628,Z 387.95,A -85,B 0,C 180,E1 -24925.475,E2 -24925.475} C_VEL
LIN {X 0,Y 133.714,Z 391.26,A -85,B 0,C 180,E1 -24930,E2 -24930} C_VEL
LIN {X 0,Y 133.567,Z 392.844,A -85,B 0,C 180,E1 -24933.016,E2 -24933.016} C_VEL
LIN {X 0,Y 133.876,Z 394.801,A -85,B 0,C 180,E1 -24939.061,E2 -24939.061} C_VEL
LIN {X 0,Y 135.446,Z 395.194,A -85,B 0,C 180,E1 -24945.036,E2 -24945.036} C_VEL
LIN {X 0,Y 138.427,Z 394.098,A -85,B 0,C 180,E1 -24950.817,E2 -24950.817} C_VEL
LIN {X 0,Y 141.475,Z 392.406,A -85,B 0,C 180,E1 -24954.651,E2 -24954.651} C_VEL
LIN {X 0,Y 142.9,Z 391.176,A -85,B 0,C 180,E1 -24956.906,E2 -24956.906} C_VEL
LIN {X 0,Y 143.953,Z 388.777,A -85,B 0,C 180,E1 -24960.737,E2 -24960.737} C_VEL
LIN {X 0,Y 145.607,Z 385.885,A -85,B 0,C 180,E1 -24964.428,E2 -24964.428} C_VEL
LIN {X 0,Y 147.887,Z 383.73,A -85,B 0,C 180,E1 -24966.382,E2 -24966.382} C_VEL
LIN {X 0,Y 153.995,Z 378.511,A -85,B 0,C 180,E1 -24969.711,E2 -24969.711} C_VEL
LIN {X 0,Y 159.245,Z 373.314,A -85,B 0,C 180,E1 -24972.3,E2 -24972.3} C_VEL
LIN {X 0,Y 166.315,Z 365.69,A -85,B 0,C 180,E1 -24975.055,E2 -24975.055} C_VEL
LIN {X 0,Y 173.672,Z 356.346,A -85,B 0,C 180,E1 -24977.604,E2 -24977.604} C_VEL
LIN {X 0,Y 180.718,Z 345.87,A -85,B 0,C 180,E1 -24979.746,E2 -24979.746} C_VEL
LIN {X 0,Y 186.811,Z 335.128,A -85,B 0,C 180,E1 -24981.317,E2 -24981.317} C_VEL
LIN {X 0,Y 192.368,Z 323.219,A -85,B 0,C 180,E1 -24982.618,E2 -24982.618} C_VEL
LIN {X 0,Y 197.037,Z 310.601,A -85,B 0,C 180,E1 -24983.603,E2 -24983.603} C_VEL
LIN {X 0,Y 200.643,Z 297.372,A -85,B 0,C 180,E1 -24984.333,E2 -24984.333} C_VEL
LIN {X 0,Y 203.082,Z 283.806,A -85,B 0,C 180,E1 -24984.86,E2 -24984.86} C_VEL
LIN {X 0,Y 203.969,Z 276.903,A -85,B 0,C 180,E1 -24985.126,E2 -24985.126} C_VEL
LIN {X 0,Y 202.666,Z 272.196,A -85,B 0,C 180,E1 -24987.37,E2 -24987.37} C_VEL
LIN {X 0,Y 201.237,Z 267.438,A -85,B 0,C 180,E1 -24990.53,E2 -24990.53} C_VEL
LIN {X 0,Y 200.272,Z 263.945,A -85,B 0,C 180,E1 -24994.357,E2 -24994.357} C_VEL
LIN {X 0,Y 200.007,Z 263.229,A -85,B 0,C 180,E1 -24997.261,E2 -24997.261} C_VEL
LIN {X 0,Y 200.535,Z 263.406,A -85,B 0,C 180,E1 -25000.856,E2 -25000.856} C_VEL
LIN {X 0,Y 202.111,Z 266.863,A -85,B 0,C 180,E1 -25005.283,E2 -25005.283} C_VEL
LIN {X 0,Y 203.811,Z 270.974,A -85,B 0,C 180,E1 -25008.195,E2 -25008.195} C_VEL
LIN {X 0,Y 204.486,Z 272.6,A -85,B 0,C 180,E1 -25009.176,E2 -25009.176} C_VEL
LIN {X 0,Y 201.71,Z 290.75,A -85,B 0,C 180,E1 -25009.827,E2 -25009.827} C_VEL
LIN {X 0,Y 198.565,Z 303.695,A -85,B 0,C 180,E1 -25010.538,E2 -25010.538} C_VEL
LIN {X 0,Y 194.333,Z 316.36,A -85,B 0,C 180,E1 -25011.551,E2 -25011.551} C_VEL
LIN {X 0,Y 189.622,Z 327.472,A -85,B 0,C 180,E1 -25012.761,E2 -25012.761} C_VEL
LIN {X 0,Y 184.444,Z 337.531,A -85,B 0,C 180,E1 -25014.204,E2 -25014.204} C_VEL
LIN {X 0,Y 177.947,Z 347.941,A -85,B 0,C 180,E1 -25016.132,E2 -25016.132} C_VEL
LIN {X 0,Y 170.934,Z 357.441,A -85,B 0,C 180,E1 -25018.492,E2 -25018.492} C_VEL
LIN {X 0,Y 164.267,Z 365.22,A -85,B 0,C 180,E1 -25021.038,E2 -25021.038} C_VEL
LIN {X 0,Y 158.028,Z 371.565,A -85,B 0,C 180,E1 -25023.824,E2 -25023.824} C_VEL
LIN {X 0,Y 151.277,Z 377.461,A -85,B 0,C 180,E1 -25027.339,E2 -25027.339} C_VEL
LIN {X 0,Y 145.251,Z 381.979,A -85,B 0,C 180,E1 -25031.158,E2 -25031.158} C_VEL
LIN {X 0,Y 139.017,Z 385.872,A -85,B 0,C 180,E1 -25036.153,E2 -25036.153} C_VEL
LIN {X 0,Y 133.984,Z 388.175,A -85,B 0,C 180,E1 -25041.54,E2 -25041.54} C_VEL
LIN {X 0,Y 131.242,Z 388.901,A -85,B 0,C 180,E1 -25045.365,E2 -25045.365} C_VEL
LIN {X 0,Y 129.056,Z 388.962,A -85,B 0,C 180,E1 -25049.391,E2 -25049.391} C_VEL
LIN {X 0,Y 127.265,Z 388.236,A -85,B 0,C 180,E1 -25054.073,E2 -25054.073} C_VEL
LIN {X 0,Y 126.206,Z 386.658,A -85,B 0,C 180,E1 -25058.777,E2 -25058.777} C_VEL
LIN {X 0,Y 125.914,Z 383.288,A -85,B 0,C 180,E1 -25064.853,E2 -25064.853} C_VEL
LIN {X 0,Y 126.329,Z 379.493,A -85,B 0,C 180,E1 -25069.662,E2 -25069.662} C_VEL
LIN {X 0,Y 127.145,Z 374.814,A -85,B 0,C 180,E1 -25074.211,E2 -25074.211} C_VEL
LIN {X 0,Y 128.435,Z 368.989,A -85,B 0,C 180,E1 -25078.681,E2 -25078.681} C_VEL
LIN {X 0,Y 130.015,Z 362.555,A -85,B 0,C 180,E1 -25082.648,E2 -25082.648} C_VEL
LIN {X 0,Y 132.356,Z 353.8,A -85,B 0,C 180,E1 -25086.946,E2 -25086.946} C_VEL
LIN {X 0,Y 134.884,Z 344.667,A -85,B 0,C 180,E1 -25090.486,E2 -25090.486} C_VEL
LIN {X 0,Y 137.666,Z 333.884,A -85,B 0,C 180,E1 -25093.754,E2 -25093.754} C_VEL
LIN {X 0,Y 140.504,Z 321.615,A -85,B 0,C 180,E1 -25096.625,E2 -25096.625} C_VEL
LIN {X 0,Y 143.002,Z 308.915,A -85,B 0,C 180,E1 -25098.818,E2 -25098.818} C_VEL
LIN {X 0,Y 145.005,Z 295.564,A -85,B 0,C 180,E1 -25100.498,E2 -25100.498} C_VEL
LIN {X 0,Y 146.502,Z 281.958,A -85,B 0,C 180,E1 -25101.596,E2 -25101.596} C_VEL
LIN {X 0,Y 150.04,Z 233.247,A -85,B 0,C 180,E1 -25104.209,E2 -25104.209} C_VEL
LIN {X 0,Y 146.374,Z 222.649,A -85,B 0,C 180,E1 -25105.698,E2 -25105.698} C_VEL
LIN {X 0,Y 140.226,Z 208.347,A -85,B 0,C 180,E1 -25108.134,E2 -25108.134} C_VEL
LIN {X 0,Y 131.9,Z 191.534,A -85,B 0,C 180,E1 -25111.625,E2 -25111.625} C_VEL
LIN {X 0,Y 130.052,Z 188.783,A -85,B 0,C 180,E1 -25112.401,E2 -25112.401} C_VEL
LIN {X 0,Y 129.68,Z 187.338,A -85,B 0,C 180,E1 -25112.757,E2 -25112.757} C_VEL
LIN {X 0,Y 129.466,Z 187.362,A -85,B 0,C 180,E1 -25119.373,E2 -25119.373} C_VEL
LIN {X 0,Y 129.294,Z 187.381,A -85,B 0,C 180,E1 -25122.558,E2 -25122.558} C_VEL
LIN {X 0,Y 129.078,Z 187.408,A -85,B 0,C 180,E1 -25129.068,E2 -25129.068} C_VEL
LIN {X 0,Y 129.031,Z 187.412,A -85,B 0,C 180,E1 -25132.413,E2 -25132.413} C_VEL
LIN {X 0,Y 128.996,Z 187.41,A -85,B 0,C 180,E1 -25139.363,E2 -25139.363} C_VEL
LIN {X 0,Y 128.953,Z 187.418,A -85,B 0,C 180,E1 -25145.166,E2 -25145.166} C_VEL
LIN {X 0,Y 128.919,Z 187.413,A -85,B 0,C 180,E1 -25150.857,E2 -25150.857} C_VEL
LIN {X 0,Y 128.909,Z 187.411,A -85,B 0,C 180,E1 -25155.133,E2 -25155.133} C_VEL
LIN {X 0,Y 128.931,Z 187.424,A -85,B 0,C 180,E1 -25159.741,E2 -25159.741} C_VEL
LIN {X 0,Y 128.953,Z 187.401,A -85,B 0,C 180,E1 -25164.836,E2 -25164.836} C_VEL
LIN {X 0,Y 128.998,Z 187.407,A -85,B 0,C 180,E1 -25170.657,E2 -25170.657} C_VEL
LIN {X 0,Y 129.065,Z 187.397,A -85,B 0,C 180,E1 -25177.774,E2 -25177.774} C_VEL
LIN {X 0,Y 129.142,Z 187.381,A -85,B 0,C 180,E1 -25184.212,E2 -25184.212} C_VEL
LIN {X 0,Y 129.341,Z 187.37,A -85,B 0,C 180,E1 -25187.975,E2 -25187.975} C_VEL
LIN {X 0,Y 129.458,Z 187.351,A -85,B 0,C 180,E1 -25190.628,E2 -25190.628} C_VEL
LIN {X 0,Y 130.064,Z 187.279,A -85,B 0,C 180,E1 -25200.001,E2 -25200.001} C_VEL
LIN {X 0,Y 129.459,Z 187.351,A -85,B 0,C 180,E1 -25209.374,E2 -25209.374} C_VEL
LIN {X 0,Y 129.296,Z 187.379,A -85,B 0,C 180,E1 -25212.559,E2 -25212.559} C_VEL
LIN {X 0,Y 129.079,Z 187.403,A -85,B 0,C 180,E1 -25219.069,E2 -25219.069} C_VEL
LIN {X 0,Y 129.033,Z 187.411,A -85,B 0,C 180,E1 -25222.414,E2 -25222.414} C_VEL
LIN {X 0,Y 128.981,Z 187.419,A -85,B 0,C 180,E1 -25229.368,E2 -25229.368} C_VEL
LIN {X 0,Y 128.955,Z 187.403,A -85,B 0,C 180,E1 -25235.166,E2 -25235.166} C_VEL
LIN {X 0,Y 128.918,Z 187.425,A -85,B 0,C 180,E1 -25240.634,E2 -25240.634} C_VEL
LIN {X 0,Y 129.981,Z 190.375,A -85,B 0,C 180,E1 -25241.223,E2 -25241.223} C_VEL
LIN {X 0,Y 131.404,Z 192.665,A -85,B 0,C 180,E1 -25241.828,E2 -25241.828} C_VEL
LIN {X 0,Y 136.706,Z 202.388,A -85,B 0,C 180,E1 -25244.051,E2 -25244.051} C_VEL
LIN {X 0,Y 142.659,Z 217.69,A -85,B 0,C 180,E1 -25246.638,E2 -25246.638} C_VEL
LIN {X 0,Y 148.614,Z 235.478,A -85,B 0,C 180,E1 -25249.171,E2 -25249.171} C_VEL
LIN {X 0,Y 149.415,Z 246.504,A -85,B 0,C 180,E1 -25250.069,E2 -25250.069} C_VEL
LIN {X 0,Y 146.07,Z 292.504,A -85,B 0,C 180,E1 -25252.596,E2 -25252.596} C_VEL
LIN {X 0,Y 144.396,Z 306.1,A -85,B 0,C 180,E1 -25253.833,E2 -25253.833} C_VEL
LIN {X 0,Y 142.186,Z 319.134,A -85,B 0,C 180,E1 -25255.575,E2 -25255.575} C_VEL
LIN {X 0,Y 139.292,Z 332.205,A -85,B 0,C 180,E1 -25258.01,E2 -25258.01} C_VEL
LIN {X 0,Y 136.53,Z 343.202,A -85,B 0,C 180,E1 -25260.725,E2 -25260.725} C_VEL
LIN {X 0,Y 133.584,Z 354.2,A -85,B 0,C 180,E1 -25264.292,E2 -25264.292} C_VEL
LIN {X 0,Y 131.247,Z 363.109,A -85,B 0,C 180,E1 -25267.986,E2 -25267.986} C_VEL
LIN {X 0,Y 129.336,Z 370.467,A -85,B 0,C 180,E1 -25271.793,E2 -25271.793} C_VEL
LIN {X 0,Y 127.737,Z 377.668,A -85,B 0,C 180,E1 -25276.477,E2 -25276.477} C_VEL
LIN {X 0,Y 126.981,Z 382.526,A -85,B 0,C 180,E1 -25280.442,E2 -25280.442} C_VEL
LIN {X 0,Y 126.566,Z 387.145,A -85,B 0,C 180,E1 -25285.222,E2 -25285.222} C_VEL
LIN {X 0,Y 126.635,Z 390.598,A -85,B 0,C 180,E1 -25289.999,E2 -25289.999} C_VEL
LIN {X 0,Y 126.493,Z 392.279,A -85,B 0,C 180,E1 -25293.184,E2 -25293.184} C_VEL
LIN {X 0,Y 126.865,Z 394.399,A -85,B 0,C 180,E1 -25299.566,E2 -25299.566} C_VEL
LIN {X 0,Y 128.585,Z 395.024,A -85,B 0,C 180,E1 -25305.859,E2 -25305.859} C_VEL
LIN {X 0,Y 131.815,Z 394.112,A -85,B 0,C 180,E1 -25311.913,E2 -25311.913} C_VEL
LIN {X 0,Y 136.646,Z 391.73,A -85,B 0,C 180,E1 -25317.573,E2 -25317.573} C_VEL
LIN {X 0,Y 141.122,Z 388.893,A -85,B 0,C 180,E1 -25321.527,E2 -25321.527} C_VEL
LIN {X 0,Y 146.071,Z 385.137,A -85,B 0,C 180,E1 -25325.264,E2 -25325.264} C_VEL
LIN {X 0,Y 147.887,Z 383.73,A -85,B 0,C 180,E1 -25326.382,E2 -25326.382} C_VEL
LIN {X 0,Y 150.349,Z 381.447,A -85,B 0,C 180,E1 -25328.252,E2 -25328.252} C_VEL
LIN {X 0,Y 153.173,Z 377.473,A -85,B 0,C 180,E1 -25331.516,E2 -25331.516} C_VEL
LIN {X 0,Y 156.312,Z 372.865,A -85,B 0,C 180,E1 -25334.533,E2 -25334.533} C_VEL
LIN {X 0,Y 159.148,Z 369.597,A -85,B 0,C 180,E1 -25335.976,E2 -25335.976} C_VEL
LIN {X 0,Y 166.507,Z 361.461,A -85,B 0,C 180,E1 -25338.519,E2 -25338.519} C_VEL
LIN {X 0,Y 174.363,Z 351.193,A -85,B 0,C 180,E1 -25340.886,E2 -25340.886} C_VEL
LIN {X 0,Y 180.488,Z 341.757,A -85,B 0,C 180,E1 -25342.501,E2 -25342.501} C_VEL
LIN {X 0,Y 186.87,Z 330.088,A -85,B 0,C 180,E1 -25343.957,E2 -25343.957} C_VEL
LIN {X 0,Y 191.914,Z 318.735,A -85,B 0,C 180,E1 -25345.021,E2 -25345.021} C_VEL
LIN {X 0,Y 196.15,Z 306.684,A -85,B 0,C 180,E1 -25345.847,E2 -25345.847} C_VEL
LIN {X 0,Y 199.605,Z 293.169,A -85,B 0,C 180,E1 -25346.47,E2 -25346.47} C_VEL
LIN {X 0,Y 201.607,Z 280.986,A -85,B 0,C 180,E1 -25346.908,E2 -25346.908} C_VEL
LIN {X 0,Y 200.454,Z 276.634,A -85,B 0,C 180,E1 -25349.299,E2 -25349.299} C_VEL
LIN {X 0,Y 199.741,Z 273.841,A -85,B 0,C 180,E1 -25351.389,E2 -25351.389} C_VEL
LIN {X 0,Y 199.06,Z 270.689,A -85,B 0,C 180,E1 -25354.933,E2 -25354.933} C_VEL
LIN {X 0,Y 199.098,Z 270.183,A -85,B 0,C 180,E1 -25359.329,E2 -25359.329} C_VEL
LIN {X 0,Y 199.356,Z 270.466,A -85,B 0,C 180,E1 -25360.738,E2 -25360.738} C_VEL
LIN {X 0,Y 200.685,Z 273.61,A -85,B 0,C 180,E1 -25364.772,E2 -25364.772} C_VEL
LIN {X 0,Y 202.008,Z 277.198,A -85,B 0,C 180,E1 -25367.344,E2 -25367.344} C_VEL
LIN {X 0,Y 199.564,Z 292.214,A -85,B 0,C 180,E1 -25367.94,E2 -25367.94} C_VEL
LIN {X 0,Y 196.355,Z 304.525,A -85,B 0,C 180,E1 -25368.602,E2 -25368.602} C_VEL
LIN {X 0,Y 191.925,Z 317.115,A -85,B 0,C 180,E1 -25369.583,E2 -25369.583} C_VEL
LIN {X 0,Y 186.832,Z 328.493,A -85,B 0,C 180,E1 -25370.8,E2 -25370.8} C_VEL
LIN {X 0,Y 180.487,Z 339.923,A -85,B 0,C 180,E1 -25372.447,E2 -25372.447} C_VEL
LIN {X 0,Y 173.312,Z 350.647,A -85,B 0,C 180,E1 -25374.493,E2 -25374.493} C_VEL
LIN {X 0,Y 166.925,Z 358.701,A -85,B 0,C 180,E1 -25376.551,E2 -25376.551} C_VEL
LIN {X 0,Y 158.768,Z 367.394,A -85,B 0,C 180,E1 -25379.539,E2 -25379.539} C_VEL
LIN {X 0,Y 151.674,Z 373.889,A -85,B 0,C 180,E1 -25382.655,E2 -25382.655} C_VEL
LIN {X 0,Y 146.029,Z 378.367,A -85,B 0,C 180,E1 -25385.522,E2 -25385.522} C_VEL
LIN {X 0,Y 140.892,Z 381.967,A -85,B 0,C 180,E1 -25388.605,E2 -25388.605} C_VEL
LIN {X 0,Y 134.04,Z 385.917,A -85,B 0,C 180,E1 -25393.646,E2 -25393.646} C_VEL
LIN {X 0,Y 128.423,Z 388.318,A -85,B 0,C 180,E1 -25399.167,E2 -25399.167} C_VEL
LIN {X 0,Y 124.092,Z 389.219,A -85,B 0,C 180,E1 -25405.022,E2 -25405.022} C_VEL
LIN {X 0,Y 120.926,Z 388.686,A -85,B 0,C 180,E1 -25411.536,E2 -25411.536} C_VEL
LIN {X 0,Y 119.605,Z 387.452,A -85,B 0,C 180,E1 -25415.985,E2 -25415.985} C_VEL
LIN {X 0,Y 118.914,Z 385.52,A -85,B 0,C 180,E1 -25420.549,E2 -25420.549} C_VEL
LIN {X 0,Y 118.833,Z 382.745,A -85,B 0,C 180,E1 -25425.209,E2 -25425.209} C_VEL
LIN {X 0,Y 119.277,Z 378.969,A -85,B 0,C 180,E1 -25429.992,E2 -25429.992} C_VEL
LIN {X 0,Y 120.183,Z 373.933,A -85,B 0,C 180,E1 -25434.951,E2 -25434.951} C_VEL
LIN {X 0,Y 121.694,Z 367.347,A -85,B 0,C 180,E1 -25440.025,E2 -25440.025} C_VEL
LIN {X 0,Y 123.97,Z 358.804,A -85,B 0,C 180,E1 -25445.099,E2 -25445.099} C_VEL
LIN {X 0,Y 126.645,Z 349.451,A -85,B 0,C 180,E1 -25449.427,E2 -25449.427} C_VEL
LIN {X 0,Y 129.444,Z 339.419,A -85,B 0,C 180,E1 -25453.033,E2 -25453.033} C_VEL
LIN {X 0,Y 132.385,Z 328.127,A -85,B 0,C 180,E1 -25456.179,E2 -25456.179} C_VEL
LIN {X 0,Y 135.031,Z 316.045,A -85,B 0,C 180,E1 -25458.766,E2 -25458.766} C_VEL
LIN {X 0,Y 137.407,Z 303.564,A -85,B 0,C 180,E1 -25460.712,E2 -25460.712} C_VEL
LIN {X 0,Y 139.246,Z 290.161,A -85,B 0,C 180,E1 -25462.206,E2 -25462.206} C_VEL
LIN {X 0,Y 140.748,Z 273.954,A -85,B 0,C 180,E1 -25463.276,E2 -25463.276} C_VEL
LIN {X 0,Y 143.659,Z 234.63,A -85,B 0,C 180,E1 -25465.449,E2 -25465.449} C_VEL
LIN {X 0,Y 140.351,Z 225.194,A -85,B 0,C 180,E1 -25466.866,E2 -25466.866} C_VEL
LIN {X 0,Y 134.386,Z 211.333,A -85,B 0,C 180,E1 -25469.363,E2 -25469.363} C_VEL
LIN {X 0,Y 127.056,Z 196.278,A -85,B 0,C 180,E1 -25472.687,E2 -25472.687} C_VEL
LIN {X 0,Y 124.112,Z 191.894,A -85,B 0,C 180,E1 -25473.997,E2 -25473.997} C_VEL
LIN {X 0,Y 122.72,Z 189.474,A -85,B 0,C 180,E1 -25474.671,E2 -25474.671} C_VEL
LIN {X 0,Y 122.455,Z 188.238,A -85,B 0,C 180,E1 -25474.939,E2 -25474.939} C_VEL
LIN {X 0,Y 122.392,Z 188.242,A -85,B 0,C 180,E1 -25479.92,E2 -25479.92} C_VEL
LIN {X 0,Y 122.183,Z 188.266,A -85,B 0,C 180,E1 -25483.302,E2 -25483.302} C_VEL
LIN {X 0,Y 121.982,Z 188.287,A -85,B 0,C 180,E1 -25490.224,E2 -25490.224} C_VEL
LIN {X 0,Y 121.908,Z 188.298,A -85,B 0,C 180,E1 -25493.801,E2 -25493.801} C_VEL
LIN {X 0,Y 121.912,Z 188.288,A -85,B 0,C 180,E1 -25500.152,E2 -25500.152} C_VEL
LIN {X 0,Y 121.877,Z 188.302,A -85,B 0,C 180,E1 -25506.169,E2 -25506.169} C_VEL
LIN {X 0,Y 121.86,Z 188.289,A -85,B 0,C 180,E1 -25511.434,E2 -25511.434} C_VEL
LIN {X 0,Y 121.86,Z 188.303,A -85,B 0,C 180,E1 -25518.568,E2 -25518.568} C_VEL
LIN {X 0,Y 121.904,Z 188.278,A -85,B 0,C 180,E1 -25524.796,E2 -25524.796} C_VEL
LIN {X 0,Y 121.913,Z 188.285,A -85,B 0,C 180,E1 -25529.85,E2 -25529.85} C_VEL
LIN {X 0,Y 121.976,Z 188.283,A -85,B 0,C 180,E1 -25537.202,E2 -25537.202} C_VEL
LIN {X 0,Y 122.055,Z 188.255,A -85,B 0,C 180,E1 -25543.269,E2 -25543.269} C_VEL
LIN {X 0,Y 122.285,Z 188.248,A -85,B 0,C 180,E1 -25547.695,E2 -25547.695} C_VEL
LIN {X 0,Y 122.387,Z 188.234,A -85,B 0,C 180,E1 -25550.081,E2 -25550.081} C_VEL
LIN {X 0,Y 122.55,Z 188.196,A -85,B 0,C 180,E1 -25556.714,E2 -25556.714} C_VEL
LIN {X 0,Y 123.017,Z 188.157,A -85,B 0,C 180,E1 -25560.001,E2 -25560.001} C_VEL
LIN {X 0,Y 122.399,Z 188.217,A -85,B 0,C 180,E1 -25566.596,E2 -25566.596} C_VEL
LIN {X 0,Y 122.388,Z 188.233,A -85,B 0,C 180,E1 -25569.921,E2 -25569.921} C_VEL
LIN {X 0,Y 122.185,Z 188.265,A -85,B 0,C 180,E1 -25573.303,E2 -25573.303} C_VEL
LIN {X 0,Y 121.985,Z 188.291,A -85,B 0,C 180,E1 -25580.225,E2 -25580.225} C_VEL
LIN {X 0,Y 121.91,Z 188.292,A -85,B 0,C 180,E1 -25583.801,E2 -25583.801} C_VEL
LIN {X 0,Y 121.904,Z 188.295,A -85,B 0,C 180,E1 -25590.143,E2 -25590.143} C_VEL
LIN {X 0,Y 121.88,Z 188.293,A -85,B 0,C 180,E1 -25596.169,E2 -25596.169} C_VEL
LIN {X 0,Y 121.827,Z 188.31,A -85,B 0,C 180,E1 -25598.394,E2 -25598.394} C_VEL
LIN {X 0,Y 122.81,Z 191.072,A -85,B 0,C 180,E1 -25599.015,E2 -25599.015} C_VEL
LIN {X 0,Y 124.382,Z 193.472,A -85,B 0,C 180,E1 -25599.74,E2 -25599.74} C_VEL
LIN {X 0,Y 131.158,Z 205.821,A -85,B 0,C 180,E1 -25602.833,E2 -25602.833} C_VEL
LIN {X 0,Y 137.256,Z 221.782,A -85,B 0,C 180,E1 -25605.666,E2 -25605.666} C_VEL
LIN {X 0,Y 142.433,Z 237.515,A -85,B 0,C 180,E1 -25608.008,E2 -25608.008} C_VEL
LIN {X 0,Y 143.115,Z 246.377,A -85,B 0,C 180,E1 -25608.787,E2 -25608.787} C_VEL
LIN {X 0,Y 139.581,Z 292.995,A -85,B 0,C 180,E1 -25611.458,E2 -25611.458} C_VEL
LIN {X 0,Y 137.826,Z 306.36,A -85,B 0,C 180,E1 -25612.733,E2 -25612.733} C_VEL
LIN {X 0,Y 135.742,Z 318.248,A -85,B 0,C 180,E1 -25614.376,E2 -25614.376} C_VEL
LIN {X 0,Y 132.923,Z 330.7,A -85,B 0,C 180,E1 -25616.732,E2 -25616.732} C_VEL
LIN {X 0,Y 129.89,Z 342.425,A -85,B 0,C 180,E1 -25619.694,E2 -25619.694} C_VEL
LIN {X 0,Y 127.147,Z 352.346,A -85,B 0,C 180,E1 -25622.97,E2 -25622.97} C_VEL
LIN {X 0,Y 124.657,Z 361.344,A -85,B 0,C 180,E1 -25626.756,E2 -25626.756} C_VEL
LIN {X 0,Y 122.611,Z 368.948,A -85,B 0,C 180,E1 -25630.756,E2 -25630.756} C_VEL
LIN {X 0,Y 120.82,Z 376.382,A -85,B 0,C 180,E1 -25635.687,E2 -25635.687} C_VEL
LIN {X 0,Y 119.988,Z 381.409,A -85,B 0,C 180,E1 -25639.879,E2 -25639.879} C_VEL
LIN {X 0,Y 119.511,Z 386.227,A -85,B 0,C 180,E1 -25644.939,E2 -25644.939} C_VEL
LIN {X 0,Y 119.567,Z 389.863,A -85,B 0,C 180,E1 -25649.999,E2 -25649.999} C_VEL
LIN {X 0,Y 119.421,Z 391.669,A -85,B 0,C 180,E1 -25653.373,E2 -25653.373} C_VEL
LIN {X 0,Y 119.488,Z 393.045,A -85,B 0,C 180,E1 -25656.755,E2 -25656.755} C_VEL
LIN {X 0,Y 120.632,Z 394.57,A -85,B 0,C 180,E1 -25663.475,E2 -25663.475} C_VEL
LIN {X 0,Y 123.239,Z 394.638,A -85,B 0,C 180,E1 -25670.008,E2 -25670.008} C_VEL
LIN {X 0,Y 127.66,Z 393.215,A -85,B 0,C 180,E1 -25676.13,E2 -25676.13} C_VEL
LIN {X 0,Y 133.483,Z 390.274,A -85,B 0,C 180,E1 -25681.769,E2 -25681.769} C_VEL
LIN {X 0,Y 138.79,Z 386.857,A -85,B 0,C 180,E1 -25685.883,E2 -25685.883} C_VEL
LIN {X 0,Y 144.339,Z 382.826,A -85,B 0,C 180,E1 -25689.269,E2 -25689.269} C_VEL
LIN {X 0,Y 150.795,Z 377.507,A -85,B 0,C 180,E1 -25692.514,E2 -25692.514} C_VEL
LIN {X 0,Y 156.535,Z 372.181,A -85,B 0,C 180,E1 -25695.001,E2 -25695.001} C_VEL
LIN {X 0,Y 159.148,Z 369.597,A -85,B 0,C 180,E1 -25695.976,E2 -25695.976} C_VEL
LIN {X 0,Y 162.072,Z 366.197,A -85,B 0,C 180,E1 -25697.338,E2 -25697.338} C_VEL
LIN {X 0,Y 165.775,Z 360.531,A -85,B 0,C 180,E1 -25699.882,E2 -25699.882} C_VEL
LIN {X 0,Y 169.491,Z 354.509,A -85,B 0,C 180,E1 -25702.236,E2 -25702.236} C_VEL
LIN {X 0,Y 172.328,Z 350.385,A -85,B 0,C 180,E1 -25703.291,E2 -25703.291} C_VEL
LIN {X 0,Y 179.25,Z 340.008,A -85,B 0,C 180,E1 -25704.929,E2 -25704.929} C_VEL
LIN {X 0,Y 185.858,Z 327.975,A -85,B 0,C 180,E1 -25706.293,E2 -25706.293} C_VEL
LIN {X 0,Y 191.107,Z 316.081,A -85,B 0,C 180,E1 -25707.269,E2 -25707.269} C_VEL
LIN {X 0,Y 195.384,Z 303.359,A -85,B 0,C 180,E1 -25708.016,E2 -25708.016} C_VEL
LIN {X 0,Y 198.669,Z 289.595,A -85,B 0,C 180,E1 -25708.585,E2 -25708.585} C_VEL
LIN {X 0,Y 199.37,Z 285.08,A -85,B 0,C 180,E1 -25708.796,E2 -25708.796} C_VEL
LIN {X 0,Y 198.415,Z 280.638,A -85,B 0,C 180,E1 -25711.839,E2 -25711.839} C_VEL
LIN {X 0,Y 197.889,Z 277.716,A -85,B 0,C 180,E1 -25715.1,E2 -25715.1} C_VEL
LIN {X 0,Y 197.942,Z 277.168,A -85,B 0,C 180,E1 -25719.202,E2 -25719.202} C_VEL
LIN {X 0,Y 198.181,Z 277.507,A -85,B 0,C 180,E1 -25720.62,E2 -25720.62} C_VEL
LIN {X 0,Y 199.319,Z 280.462,A -85,B 0,C 180,E1 -25724.365,E2 -25724.365} C_VEL
LIN {X 0,Y 199.797,Z 281.995,A -85,B 0,C 180,E1 -25725.559,E2 -25725.559} C_VEL
LIN {X 0,Y 196.853,Z 296.649,A -85,B 0,C 180,E1 -25726.121,E2 -25726.121} C_VEL
LIN {X 0,Y 193.009,Z 309.552,A -85,B 0,C 180,E1 -25726.899,E2 -25726.899} C_VEL
LIN {X 0,Y 188.257,Z 321.457,A -85,B 0,C 180,E1 -25727.893,E2 -25727.893} C_VEL
LIN {X 0,Y 182.708,Z 332.589,A -85,B 0,C 180,E1 -25729.161,E2 -25729.161} C_VEL
LIN {X 0,Y 176.071,Z 343.441,A -85,B 0,C 180,E1 -25730.812,E2 -25730.812} C_VEL
LIN {X 0,Y 168.648,Z 353.427,A -85,B 0,C 180,E1 -25732.817,E2 -25732.817} C_VEL
LIN {X 0,Y 161.624,Z 361.514,A -85,B 0,C 180,E1 -25735.01,E2 -25735.01} C_VEL
LIN {X 0,Y 153.213,Z 369.72,A -85,B 0,C 180,E1 -25738.026,E2 -25738.026} C_VEL
LIN {X 0,Y 145.224,Z 376.25,A -85,B 0,C 180,E1 -25741.459,E2 -25741.459} C_VEL
LIN {X 0,Y 139.051,Z 380.552,A -85,B 0,C 180,E1 -25744.63,E2 -25744.63} C_VEL
LIN {X 0,Y 131.719,Z 384.831,A -85,B 0,C 180,E1 -25749.21,E2 -25749.21} C_VEL
LIN {X 0,Y 127.143,Z 386.975,A -85,B 0,C 180,E1 -25752.773,E2 -25752.773} C_VEL
LIN {X 0,Y 123.132,Z 388.463,A -85,B 0,C 180,E1 -25756.58,E2 -25756.58} C_VEL
LIN {X 0,Y 119.694,Z 389.257,A -85,B 0,C 180,E1 -25760.626,E2 -25760.626} C_VEL
LIN {X 0,Y 116.596,Z 389.432,A -85,B 0,C 180,E1 -25765.295,E2 -25765.295} C_VEL
LIN {X 0,Y 114.12,Z 388.785,A -85,B 0,C 180,E1 -25770.44,E2 -25770.44} C_VEL
LIN {X 0,Y 112.524,Z 387.26,A -85,B 0,C 180,E1 -25775.715,E2 -25775.715} C_VEL
LIN {X 0,Y 111.783,Z 384.873,A -85,B 0,C 180,E1 -25781.023,E2 -25781.023} C_VEL
LIN {X 0,Y 111.764,Z 381.646,A -85,B 0,C 180,E1 -25786.236,E2 -25786.236} C_VEL
LIN {X 0,Y 112.348,Z 377.575,A -85,B 0,C 180,E1 -25791.278,E2 -25791.278} C_VEL
LIN {X 0,Y 113.583,Z 371.589,A -85,B 0,C 180,E1 -25796.981,E2 -25796.981} C_VEL
LIN {X 0,Y 115.172,Z 365.179,A -85,B 0,C 180,E1 -25801.767,E2 -25801.767} C_VEL
LIN {X 0,Y 117.544,Z 356.885,A -85,B 0,C 180,E1 -25806.666,E2 -25806.666} C_VEL
LIN {X 0,Y 120.549,Z 346.681,A -85,B 0,C 180,E1 -25811.299,E2 -25811.299} C_VEL
LIN {X 0,Y 123.637,Z 335.849,A -85,B 0,C 180,E1 -25815.087,E2 -25815.087} C_VEL
LIN {X 0,Y 126.703,Z 323.935,A -85,B 0,C 180,E1 -25818.239,E2 -25818.239} C_VEL
LIN {X 0,Y 129.277,Z 312.142,A -85,B 0,C 180,E1 -25820.614,E2 -25820.614} C_VEL
LIN {X 0,Y 131.628,Z 298.969,A -85,B 0,C 180,E1 -25822.523,E2 -25822.523} C_VEL
LIN {X 0,Y 133.383,Z 284.977,A -85,B 0,C 180,E1 -25823.904,E2 -25823.904} C_VEL
LIN {X 0,Y 137.319,Z 236.799,A -85,B 0,C 180,E1 -25826.701,E2 -25826.701} C_VEL
LIN {X 0,Y 135.703,Z 231.109,A -85,B 0,C 180,E1 -25827.508,E2 -25827.508} C_VEL
LIN {X 0,Y 129.224,Z 215.563,A -85,B 0,C 180,E1 -25830.429,E2 -25830.429} C_VEL
LIN {X 0,Y 122.109,Z 200.783,A -85,B 0,C 180,E1 -25833.852,E2 -25833.852} C_VEL
LIN {X 0,Y 117.799,Z 193.91,A -85,B 0,C 180,E1 -25835.971,E2 -25835.971} C_VEL
LIN {X 0,Y 115.678,Z 190.596,A -85,B 0,C 180,E1 -25837.089,E2 -25837.089} C_VEL
LIN {X 0,Y 115.329,Z 189.123,A -85,B 0,C 180,E1 -25837.441,E2 -25837.441} C_VEL
LIN {X 0,Y 115.201,Z 189.137,A -85,B 0,C 180,E1 -25842.558,E2 -25842.558} C_VEL
LIN {X 0,Y 114.96,Z 189.165,A -85,B 0,C 180,E1 -25847.799,E2 -25847.799} C_VEL
LIN {X 0,Y 114.89,Z 189.174,A -85,B 0,C 180,E1 -25853.43,E2 -25853.43} C_VEL
LIN {X 0,Y 114.844,Z 189.162,A -85,B 0,C 180,E1 -25861.05,E2 -25861.05} C_VEL
LIN {X 0,Y 114.772,Z 189.188,A -85,B 0,C 180,E1 -25867.759,E2 -25867.759} C_VEL
LIN {X 0,Y 114.765,Z 189.164,A -85,B 0,C 180,E1 -25872.707,E2 -25872.707} C_VEL
LIN {X 0,Y 114.783,Z 189.183,A -85,B 0,C 180,E1 -25877.663,E2 -25877.663} C_VEL
LIN {X 0,Y 114.78,Z 189.178,A -85,B 0,C 180,E1 -25882.749,E2 -25882.749} C_VEL
LIN {X 0,Y 114.844,Z 189.158,A -85,B 0,C 180,E1 -25888.953,E2 -25888.953} C_VEL
LIN {X 0,Y 114.891,Z 189.167,A -85,B 0,C 180,E1 -25896.573,E2 -25896.573} C_VEL
LIN {X 0,Y 114.96,Z 189.131,A -85,B 0,C 180,E1 -25902.203,E2 -25902.203} C_VEL
LIN {X 0,Y 115.302,Z 189.118,A -85,B 0,C 180,E1 -25909.465,E2 -25909.465} C_VEL
LIN {X 0,Y 115.477,Z 189.075,A -85,B 0,C 180,E1 -25916.512,E2 -25916.512} C_VEL
LIN {X 0,Y 115.969,Z 189.035,A -85,B 0,C 180,E1 -25920.001,E2 -25920.001} C_VEL
LIN {X 0,Y 115.342,Z 189.095,A -85,B 0,C 180,E1 -25927.001,E2 -25927.001} C_VEL
LIN {X 0,Y 115.203,Z 189.134,A -85,B 0,C 180,E1 -25932.557,E2 -25932.557} C_VEL
LIN {X 0,Y 114.962,Z 189.153,A -85,B 0,C 180,E1 -25937.8,E2 -25937.8} C_VEL
LIN {X 0,Y 114.893,Z 189.167,A -85,B 0,C 180,E1 -25943.43,E2 -25943.43} C_VEL
LIN {X 0,Y 114.839,Z 189.166,A -85,B 0,C 180,E1 -25951.043,E2 -25951.043} C_VEL
LIN {X 0,Y 114.875,Z 189.329,A -85,B 0,C 180,E1 -25955.98,E2 -25955.98} C_VEL
LIN {X 0,Y 115.925,Z 192.141,A -85,B 0,C 180,E1 -25956.666,E2 -25956.666} C_VEL
LIN {X 0,Y 117.407,Z 194.46,A -85,B 0,C 180,E1 -25957.444,E2 -25957.444} C_VEL
LIN {X 0,Y 123.949,Z 205.91,A -85,B 0,C 180,E1 -25960.692,E2 -25960.692} C_VEL
LIN {X 0,Y 126.464,Z 211.31,A -85,B 0,C 180,E1 -25961.929,E2 -25961.929} C_VEL
LIN {X 0,Y 131.892,Z 225.923,A -85,B 0,C 180,E1 -25964.646,E2 -25964.646} C_VEL
LIN {X 0,Y 136.353,Z 239.876,A -85,B 0,C 180,E1 -25966.815,E2 -25966.815} C_VEL
LIN {X 0,Y 136.765,Z 247.988,A -85,B 0,C 180,E1 -25967.514,E2 -25967.514} C_VEL
LIN {X 0,Y 133.193,Z 292.717,A -85,B 0,C 180,E1 -25970.179,E2 -25970.179} C_VEL
LIN {X 0,Y 131.323,Z 306.314,A -85,B 0,C 180,E1 -25971.528,E2 -25971.528} C_VEL
LIN {X 0,Y 129.166,Z 318.132,A -85,B 0,C 180,E1 -25973.236,E2 -25973.236} C_VEL
LIN {X 0,Y 126.238,Z 330.524,A -85,B 0,C 180,E1 -25975.689,E2 -25975.689} C_VEL
LIN {X 0,Y 123.241,Z 341.726,A -85,B 0,C 180,E1 -25978.643,E2 -25978.643} C_VEL
LIN {X 0,Y 120.293,Z 351.917,A -85,B 0,C 180,E1 -25982.135,E2 -25982.135} C_VEL
LIN {X 0,Y 117.66,Z 361.145,A -85,B 0,C 180,E1 -25986.222,E2 -25986.222} C_VEL
LIN {X 0,Y 115.158,Z 370.116,A -85,B 0,C 180,E1 -25991.312,E2 -25991.312} C_VEL
LIN {X 0,Y 113.503,Z 377.283,A -85,B 0,C 180,E1 -25996.573,E2 -25996.573} C_VEL
LIN {X 0,Y 112.763,Z 382.119,A -85,B 0,C 180,E1 -26001.036,E2 -26001.036} C_VEL
LIN {X 0,Y 112.412,Z 386.725,A -85,B 0,C 180,E1 -26006.415,E2 -26006.415} C_VEL
LIN {X 0,Y 112.462,Z 389.584,A -85,B 0,C 180,E1 -26010.804,E2 -26010.804} C_VEL
LIN {X 0,Y 112.453,Z 392.472,A -85,B 0,C 180,E1 -26017.18,E2 -26017.18} C_VEL
LIN {X 0,Y 113.717,Z 394.238,A -85,B 0,C 180,E1 -26024.312,E2 -26024.312} C_VEL
LIN {X 0,Y 116.57,Z 394.482,A -85,B 0,C 180,E1 -26031.206,E2 -26031.206} C_VEL
LIN {X 0,Y 121.316,Z 393.301,A -85,B 0,C 180,E1 -26037.609,E2 -26037.609} C_VEL
LIN {X 0,Y 124.212,Z 392.158,A -85,B 0,C 180,E1 -26040.611,E2 -26040.611} C_VEL
LIN {X 0,Y 130.982,Z 388.67,A -85,B 0,C 180,E1 -26046.171,E2 -26046.171} C_VEL
LIN {X 0,Y 136.853,Z 384.99,A -85,B 0,C 180,E1 -26049.934,E2 -26049.934} C_VEL
LIN {X 0,Y 143.476,Z 380.308,A -85,B 0,C 180,E1 -26053.295,E2 -26053.295} C_VEL
LIN {X 0,Y 150.403,Z 374.523,A -85,B 0,C 180,E1 -26056.408,E2 -26056.408} C_VEL
LIN {X 0,Y 159.367,Z 366,A -85,B 0,C 180,E1 -26059.526,E2 -26059.526} C_VEL
LIN {X 0,Y 167.358,Z 356.871,A -85,B 0,C 180,E1 -26061.94,E2 -26061.94} C_VEL
LIN {X 0,Y 172.328,Z 350.385,A -85,B 0,C 180,E1 -26063.291,E2 -26063.291} C_VEL
LIN {X 0,Y 175.159,Z 346.115,A -85,B 0,C 180,E1 -26064.27,E2 -26064.27} C_VEL
LIN {X 0,Y 178.873,Z 339.057,A -85,B 0,C 180,E1 -26066.181,E2 -26066.181} C_VEL
LIN {X 0,Y 182.369,Z 331.59,A -85,B 0,C 180,E1 -26067.895,E2 -26067.895} C_VEL
LIN {X 0,Y 184.768,Z 326.675,A -85,B 0,C 180,E1 -26068.571,E2 -26068.571} C_VEL
LIN {X 0,Y 190.224,Z 314.341,A -85,B 0,C 180,E1 -26069.482,E2 -26069.482} C_VEL
LIN {X 0,Y 194.151,Z 302.841,A -85,B 0,C 180,E1 -26070.096,E2 -26070.096} C_VEL
LIN {X 0,Y 197.381,Z 289.749,A -85,B 0,C 180,E1 -26070.603,E2 -26070.603} C_VEL
LIN {X 0,Y 196.97,Z 287.192,A -85,B 0,C 180,E1 -26072.509,E2 -26072.509} C_VEL
LIN {X 0,Y 196.659,Z 284.513,A -85,B 0,C 180,E1 -26075.737,E2 -26075.737} C_VEL
LIN {X 0,Y 196.929,Z 284.31,A -85,B 0,C 180,E1 -26080.151,E2 -26080.151} C_VEL
LIN {X 0,Y 197.776,Z 286.979,A -85,B 0,C 180,E1 -26083.693,E2 -26083.693} C_VEL
LIN {X 0,Y 194.713,Z 299.998,A -85,B 0,C 180,E1 -26084.245,E2 -26084.245} C_VEL
LIN {X 0,Y 190.459,Z 312.731,A -85,B 0,C 180,E1 -26085.03,E2 -26085.03} C_VEL
LIN {X 0,Y 185.294,Z 324.554,A -85,B 0,C 180,E1 -26086.046,E2 -26086.046} C_VEL
LIN {X 0,Y 178.768,Z 336.361,A -85,B 0,C 180,E1 -26087.438,E2 -26087.438} C_VEL
LIN {X 0,Y 171.793,Z 346.768,A -85,B 0,C 180,E1 -26089.055,E2 -26089.055} C_VEL
LIN {X 0,Y 165.222,Z 355.01,A -85,B 0,C 180,E1 -26090.759,E2 -26090.759} C_VEL
LIN {X 0,Y 157.52,Z 363.229,A -85,B 0,C 180,E1 -26093.016,E2 -26093.016} C_VEL
LIN {X 0,Y 150.096,Z 369.969,A -85,B 0,C 180,E1 -26095.502,E2 -26095.502} C_VEL
LIN {X 0,Y 143.027,Z 375.536,A -85,B 0,C 180,E1 -26098.27,E2 -26098.27} C_VEL
LIN {X 0,Y 136.335,Z 380.069,A -85,B 0,C 180,E1 -26101.342,E2 -26101.342} C_VEL
LIN {X 0,Y 130.316,Z 383.529,A -85,B 0,C 180,E1 -26104.639,E2 -26104.639} C_VEL
LIN {X 0,Y 122.54,Z 387.084,A -85,B 0,C 180,E1 -26109.906,E2 -26109.906} C_VEL
LIN {X 0,Y 116.577,Z 388.988,A -85,B 0,C 180,E1 -26115.301,E2 -26115.301} C_VEL
LIN {X 0,Y 111.007,Z 389.695,A -85,B 0,C 180,E1 -26122.324,E2 -26122.324} C_VEL
LIN {X 0,Y 108.37,Z 389.246,A -85,B 0,C 180,E1 -26126.996,E2 -26126.996} C_VEL
LIN {X 0,Y 106.409,Z 388.171,A -85,B 0,C 180,E1 -26131.894,E2 -26131.894} C_VEL
LIN {X 0,Y 104.829,Z 385.178,A -85,B 0,C 180,E1 -26139.559,E2 -26139.559} C_VEL
LIN {X 0,Y 104.619,Z 382.164,A -85,B 0,C 180,E1 -26144.853,E2 -26144.853} C_VEL
LIN {X 0,Y 105.156,Z 377.893,A -85,B 0,C 180,E1 -26150.589,E2 -26150.589} C_VEL
LIN {X 0,Y 106.452,Z 371.621,A -85,B 0,C 180,E1 -26156.999,E2 -26156.999} C_VEL
LIN {X 0,Y 108.468,Z 363.863,A -85,B 0,C 180,E1 -26163.029,E2 -26163.029} C_VEL
LIN {X 0,Y 111.083,Z 355.05,A -85,B 0,C 180,E1 -26168.279,E2 -26168.279} C_VEL
LIN {X 0,Y 113.864,Z 346.1,A -85,B 0,C 180,E1 -26172.436,E2 -26172.436} C_VEL
LIN {X 0,Y 116.822,Z 336.105,A -85,B 0,C 180,E1 -26176.077,E2 -26176.077} C_VEL
LIN {X 0,Y 119.632,Z 325.785,A -85,B 0,C 180,E1 -26178.994,E2 -26178.994} C_VEL
LIN {X 0,Y 122.591,Z 312.946,A -85,B 0,C 180,E1 -26181.761,E2 -26181.761} C_VEL
LIN {X 0,Y 124.817,Z 301.652,A -85,B 0,C 180,E1 -26183.535,E2 -26183.535} C_VEL
LIN {X 0,Y 126.707,Z 288.143,A -85,B 0,C 180,E1 -26185.027,E2 -26185.027} C_VEL
LIN {X 0,Y 128.395,Z 269.372,A -85,B 0,C 180,E1 -26186.286,E2 -26186.286} C_VEL
LIN {X 0,Y 131.006,Z 237.362,A -85,B 0,C 180,E1 -26188.185,E2 -26188.185} C_VEL
LIN {X 0,Y 125.686,Z 223.366,A -85,B 0,C 180,E1 -26190.802,E2 -26190.802} C_VEL
LIN {X 0,Y 117.326,Z 205.387,A -85,B 0,C 180,E1 -26195.048,E2 -26195.048} C_VEL
LIN {X 0,Y 110.748,Z 194.701,A -85,B 0,C 180,E1 -26198.65,E2 -26198.65} C_VEL
LIN {X 0,Y 108.744,Z 191.855,A -85,B 0,C 180,E1 -26199.806,E2 -26199.806} C_VEL
LIN {X 0,Y 108.271,Z 190.001,A -85,B 0,C 180,E1 -26200.282,E2 -26200.282} C_VEL
LIN {X 0,Y 107.964,Z 190.039,A -85,B 0,C 180,E1 -26205.093,E2 -26205.093} C_VEL
LIN {X 0,Y 107.856,Z 190.051,A -85,B 0,C 180,E1 -26209.015,E2 -26209.015} C_VEL
LIN {X 0,Y 107.799,Z 190.055,A -85,B 0,C 180,E1 -26214.118,E2 -26214.118} C_VEL
LIN {X 0,Y 107.769,Z 190.041,A -85,B 0,C 180,E1 -26222.033,E2 -26222.033} C_VEL
LIN {X 0,Y 107.679,Z 190.071,A -85,B 0,C 180,E1 -26228.447,E2 -26228.447} C_VEL
LIN {X 0,Y 107.664,Z 190.059,A -85,B 0,C 180,E1 -26235.894,E2 -26235.894} C_VEL
LIN {X 0,Y 107.68,Z 190.068,A -85,B 0,C 180,E1 -26241.555,E2 -26241.555} C_VEL
LIN {X 0,Y 107.781,Z 190.034,A -85,B 0,C 180,E1 -26248.559,E2 -26248.559} C_VEL
LIN {X 0,Y 107.859,Z 190.042,A -85,B 0,C 180,E1 -26256.988,E2 -26256.988} C_VEL
LIN {X 0,Y 107.857,Z 190.015,A -85,B 0,C 180,E1 -26260.987,E2 -26260.987} C_VEL
LIN {X 0,Y 108.203,Z 190.002,A -85,B 0,C 180,E1 -26268.765,E2 -26268.765} C_VEL
LIN {X 0,Y 108.281,Z 189.978,A -85,B 0,C 180,E1 -26272.543,E2 -26272.543} C_VEL
LIN {X 0,Y 108.894,Z 189.916,A -85,B 0,C 180,E1 -26280.002,E2 -26280.002} C_VEL
LIN {X 0,Y 108.282,Z 189.974,A -85,B 0,C 180,E1 -26287.46,E2 -26287.46} C_VEL
LIN {X 0,Y 108.137,Z 190.015,A -85,B 0,C 180,E1 -26292.872,E2 -26292.872} C_VEL
LIN {X 0,Y 107.859,Z 190.046,A -85,B 0,C 180,E1 -26299.016,E2 -26299.016} C_VEL
LIN {X 0,Y 107.801,Z 190.048,A -85,B 0,C 180,E1 -26304.117,E2 -26304.117} C_VEL
LIN {X 0,Y 107.772,Z 190.034,A -85,B 0,C 180,E1 -26312.626,E2 -26312.626} C_VEL
LIN {X 0,Y 107.793,Z 190.14,A -85,B 0,C 180,E1 -26313.092,E2 -26313.092} C_VEL
LIN {X 0,Y 108.751,Z 192.815,A -85,B 0,C 180,E1 -26313.811,E2 -26313.811} C_VEL
LIN {X 0,Y 110.314,Z 194.866,A -85,B 0,C 180,E1 -26314.699,E2 -26314.699} C_VEL
LIN {X 0,Y 118.399,Z 209.196,A -85,B 0,C 180,E1 -26319.188,E2 -26319.188} C_VEL
LIN {X 0,Y 121.102,Z 215.007,A -85,B 0,C 180,E1 -26320.603,E2 -26320.603} C_VEL
LIN {X 0,Y 126.112,Z 228.687,A -85,B 0,C 180,E1 -26323.294,E2 -26323.294} C_VEL
LIN {X 0,Y 130.245,Z 242.045,A -85,B 0,C 180,E1 -26325.504,E2 -26325.504} C_VEL
LIN {X 0,Y 130.509,Z 248.364,A -85,B 0,C 180,E1 -26326.073,E2 -26326.073} C_VEL
LIN {X 0,Y 126.897,Z 291.88,A -85,B 0,C 180,E1 -26328.745,E2 -26328.745} C_VEL
LIN {X 0,Y 124.887,Z 306.104,A -85,B 0,C 180,E1 -26330.199,E2 -26330.199} C_VEL
LIN {X 0,Y 122.652,Z 317.929,A -85,B 0,C 180,E1 -26331.977,E2 -26331.977} C_VEL
LIN {X 0,Y 119.59,Z 330.312,A -85,B 0,C 180,E1 -26334.526,E2 -26334.526} C_VEL
LIN {X 0,Y 116.405,Z 341.778,A -85,B 0,C 180,E1 -26337.702,E2 -26337.702} C_VEL
LIN {X 0,Y 113.409,Z 351.714,A -85,B 0,C 180,E1 -26341.297,E2 -26341.297} C_VEL
LIN {X 0,Y 110.659,Z 360.942,A -85,B 0,C 180,E1 -26345.618,E2 -26345.618} C_VEL
LIN {X 0,Y 108.455,Z 368.545,A -85,B 0,C 180,E1 -26350.11,E2 -26350.11} C_VEL
LIN {X 0,Y 106.599,Z 375.966,A -85,B 0,C 180,E1 -26355.686,E2 -26355.686} C_VEL
LIN {X 0,Y 105.752,Z 380.969,A -85,B 0,C 180,E1 -26360.436,E2 -26360.436} C_VEL
LIN {X 0,Y 105.373,Z 385.765,A -85,B 0,C 180,E1 -26366.175,E2 -26366.175} C_VEL
LIN {X 0,Y 105.426,Z 388.571,A -85,B 0,C 180,E1 -26370.428,E2 -26370.428} C_VEL
LIN {X 0,Y 105.314,Z 390.317,A -85,B 0,C 180,E1 -26373.826,E2 -26373.826} C_VEL
LIN {X 0,Y 105.912,Z 393.044,A -85,B 0,C 180,E1 -26381.482,E2 -26381.482} C_VEL
LIN {X 0,Y 108.197,Z 394.279,A -85,B 0,C 180,E1 -26388.951,E2 -26388.951} C_VEL
LIN {X 0,Y 109.96,Z 394.33,A -85,B 0,C 180,E1 -26392.549,E2 -26392.549} C_VEL
LIN {X 0,Y 115.051,Z 393.341,A -85,B 0,C 180,E1 -26399.253,E2 -26399.253} C_VEL
LIN {X 0,Y 121.648,Z 390.902,A -85,B 0,C 180,E1 -26405.29,E2 -26405.29} C_VEL
LIN {X 0,Y 126.884,Z 388.275,A -85,B 0,C 180,E1 -26409.152,E2 -26409.152} C_VEL
LIN {X 0,Y 133.728,Z 384.289,A -85,B 0,C 180,E1 -26413.093,E2 -26413.093} C_VEL
LIN {X 0,Y 140.772,Z 379.484,A -85,B 0,C 180,E1 -26416.377,E2 -26416.377} C_VEL
LIN {X 0,Y 148.276,Z 373.52,A -85,B 0,C 180,E1 -26419.319,E2 -26419.319} C_VEL
LIN {X 0,Y 156.283,Z 366.236,A -85,B 0,C 180,E1 -26421.901,E2 -26421.901} C_VEL
LIN {X 0,Y 164.594,Z 357.304,A -85,B 0,C 180,E1 -26424.219,E2 -26424.219} C_VEL
LIN {X 0,Y 172.438,Z 347.19,A -85,B 0,C 180,E1 -26426.14,E2 -26426.14} C_VEL
LIN {X 0,Y 179.122,Z 336.992,A -85,B 0,C 180,E1 -26427.517,E2 -26427.517} C_VEL
LIN {X 0,Y 184.768,Z 326.675,A -85,B 0,C 180,E1 -26428.571,E2 -26428.571} C_VEL
LIN {X 0,Y 187.1,Z 321.637,A -85,B 0,C 180,E1 -26429.196,E2 -26429.196} C_VEL
LIN {X 0,Y 190.136,Z 313.403,A -85,B 0,C 180,E1 -26430.589,E2 -26430.589} C_VEL
LIN {X 0,Y 192.651,Z 304.876,A -85,B 0,C 180,E1 -26431.87,E2 -26431.87} C_VEL
LIN {X 0,Y 194.101,Z 299.386,A -85,B 0,C 180,E1 -26432.328,E2 -26432.328} C_VEL
LIN {X 0,Y 195.359,Z 294.428,A -85,B 0,C 180,E1 -26432.554,E2 -26432.554} C_VEL
LIN {X 0,Y 195.237,Z 291.459,A -85,B 0,C 180,E1 -26435.83,E2 -26435.83} C_VEL
LIN {X 0,Y 195.428,Z 291.158,A -85,B 0,C 180,E1 -26439.649,E2 -26439.649} C_VEL
LIN {X 0,Y 195.644,Z 292.644,A -85,B 0,C 180,E1 -26441.836,E2 -26441.836} C_VEL
LIN {X 0,Y 192.201,Z 304.962,A -85,B 0,C 180,E1 -26442.406,E2 -26442.406} C_VEL
LIN {X 0,Y 187.36,Z 317.626,A -85,B 0,C 180,E1 -26443.239,E2 -26443.239} C_VEL
LIN {X 0,Y 181.697,Z 329.177,A -85,B 0,C 180,E1 -26444.29,E2 -26444.29} C_VEL
LIN {X 0,Y 174.95,Z 340.174,A -85,B 0,C 180,E1 -26445.648,E2 -26445.648} C_VEL
LIN {X 0,Y 167.495,Z 350.179,A -85,B 0,C 180,E1 -26447.273,E2 -26447.273} C_VEL
LIN {X 0,Y 159.71,Z 358.986,A -85,B 0,C 180,E1 -26449.219,E2 -26449.219} C_VEL
LIN {X 0,Y 152.143,Z 366.262,A -85,B 0,C 180,E1 -26451.364,E2 -26451.364} C_VEL
LIN {X 0,Y 143.094,Z 373.547,A -85,B 0,C 180,E1 -26454.362,E2 -26454.362} C_VEL
LIN {X 0,Y 133.595,Z 379.85,A -85,B 0,C 180,E1 -26458.196,E2 -26458.196} C_VEL
LIN {X 0,Y 126.557,Z 383.684,A -85,B 0,C 180,E1 -26461.701,E2 -26461.701} C_VEL
LIN {X 0,Y 118.338,Z 387.217,A -85,B 0,C 180,E1 -26466.82,E2 -26466.82} C_VEL
